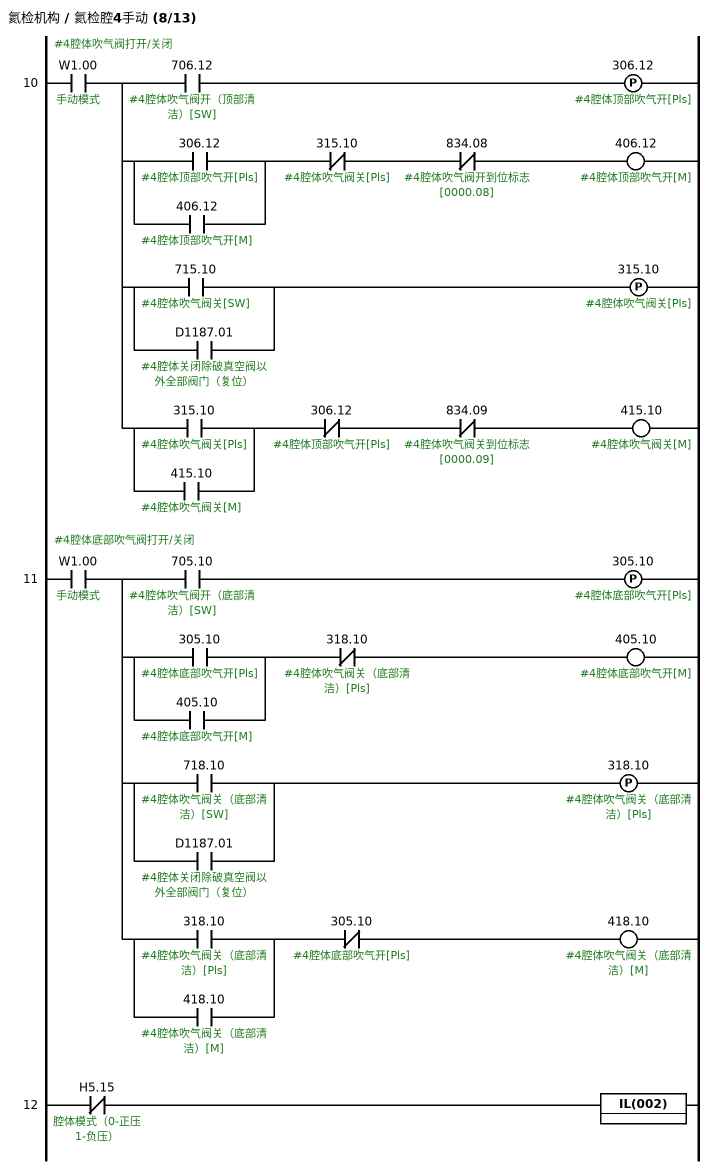
; [picture p216: 氦检机构 / 氦检腔4手动, rungs 10-12]
; rung 10: #4腔体吹气阀打开/关闭
LD W1.00  ; 手动模式
OUT TR0
AND 706.12  ; #4腔体吹气阀开（顶部清洁）[SW]
DIFU(013) 306.12  ; #4腔体顶部吹气开[Pls]
LD TR0
LD 306.12  ; #4腔体顶部吹气开[Pls]
OR 406.12  ; #4腔体顶部吹气开[M]
ANDLD
ANDNOT 315.10  ; #4腔体吹气阀关[Pls]
ANDNOT 834.08  ; #4腔体吹气阀开到位标志[0000.08]
OUT 406.12  ; #4腔体顶部吹气开[M]
LD TR0
LD 715.10  ; #4腔体吹气阀关[SW]
OR D1187.01  ; #4腔体关闭除破真空阀以外全部阀门（复位）
ANDLD
DIFU(013) 315.10  ; #4腔体吹气阀关[Pls]
LD TR0
LD 315.10  ; #4腔体吹气阀关[Pls]
OR 415.10  ; #4腔体吹气阀关[M]
ANDLD
ANDNOT 306.12  ; #4腔体顶部吹气开[Pls]
ANDNOT 834.09  ; #4腔体吹气阀关到位标志[0000.09]
OUT 415.10  ; #4腔体吹气阀关[M]
; rung 11: #4腔体底部吹气阀打开/关闭
LD W1.00  ; 手动模式
OUT TR0
AND 705.10  ; #4腔体吹气阀开（底部清洁）[SW]
DIFU(013) 305.10  ; #4腔体底部吹气开[Pls]
LD TR0
LD 305.10  ; #4腔体底部吹气开[Pls]
OR 405.10  ; #4腔体底部吹气开[M]
ANDLD
ANDNOT 318.10  ; #4腔体吹气阀关（底部清洁）[Pls]
OUT 405.10  ; #4腔体底部吹气开[M]
LD TR0
LD 718.10  ; #4腔体吹气阀关（底部清洁）[SW]
OR D1187.01  ; #4腔体关闭除破真空阀以外全部阀门（复位）
ANDLD
DIFU(013) 318.10  ; #4腔体吹气阀关（底部清洁）[Pls]
LD TR0
LD 318.10  ; #4腔体吹气阀关（底部清洁）[Pls]
OR 418.10  ; #4腔体吹气阀关（底部清洁）[M]
ANDLD
ANDNOT 305.10  ; #4腔体底部吹气开[Pls]
OUT 418.10  ; #4腔体吹气阀关（底部清洁）[M]
; rung 12
LDNOT H5.15  ; 腔体模式（0-正压 1-负压）
IL(002)

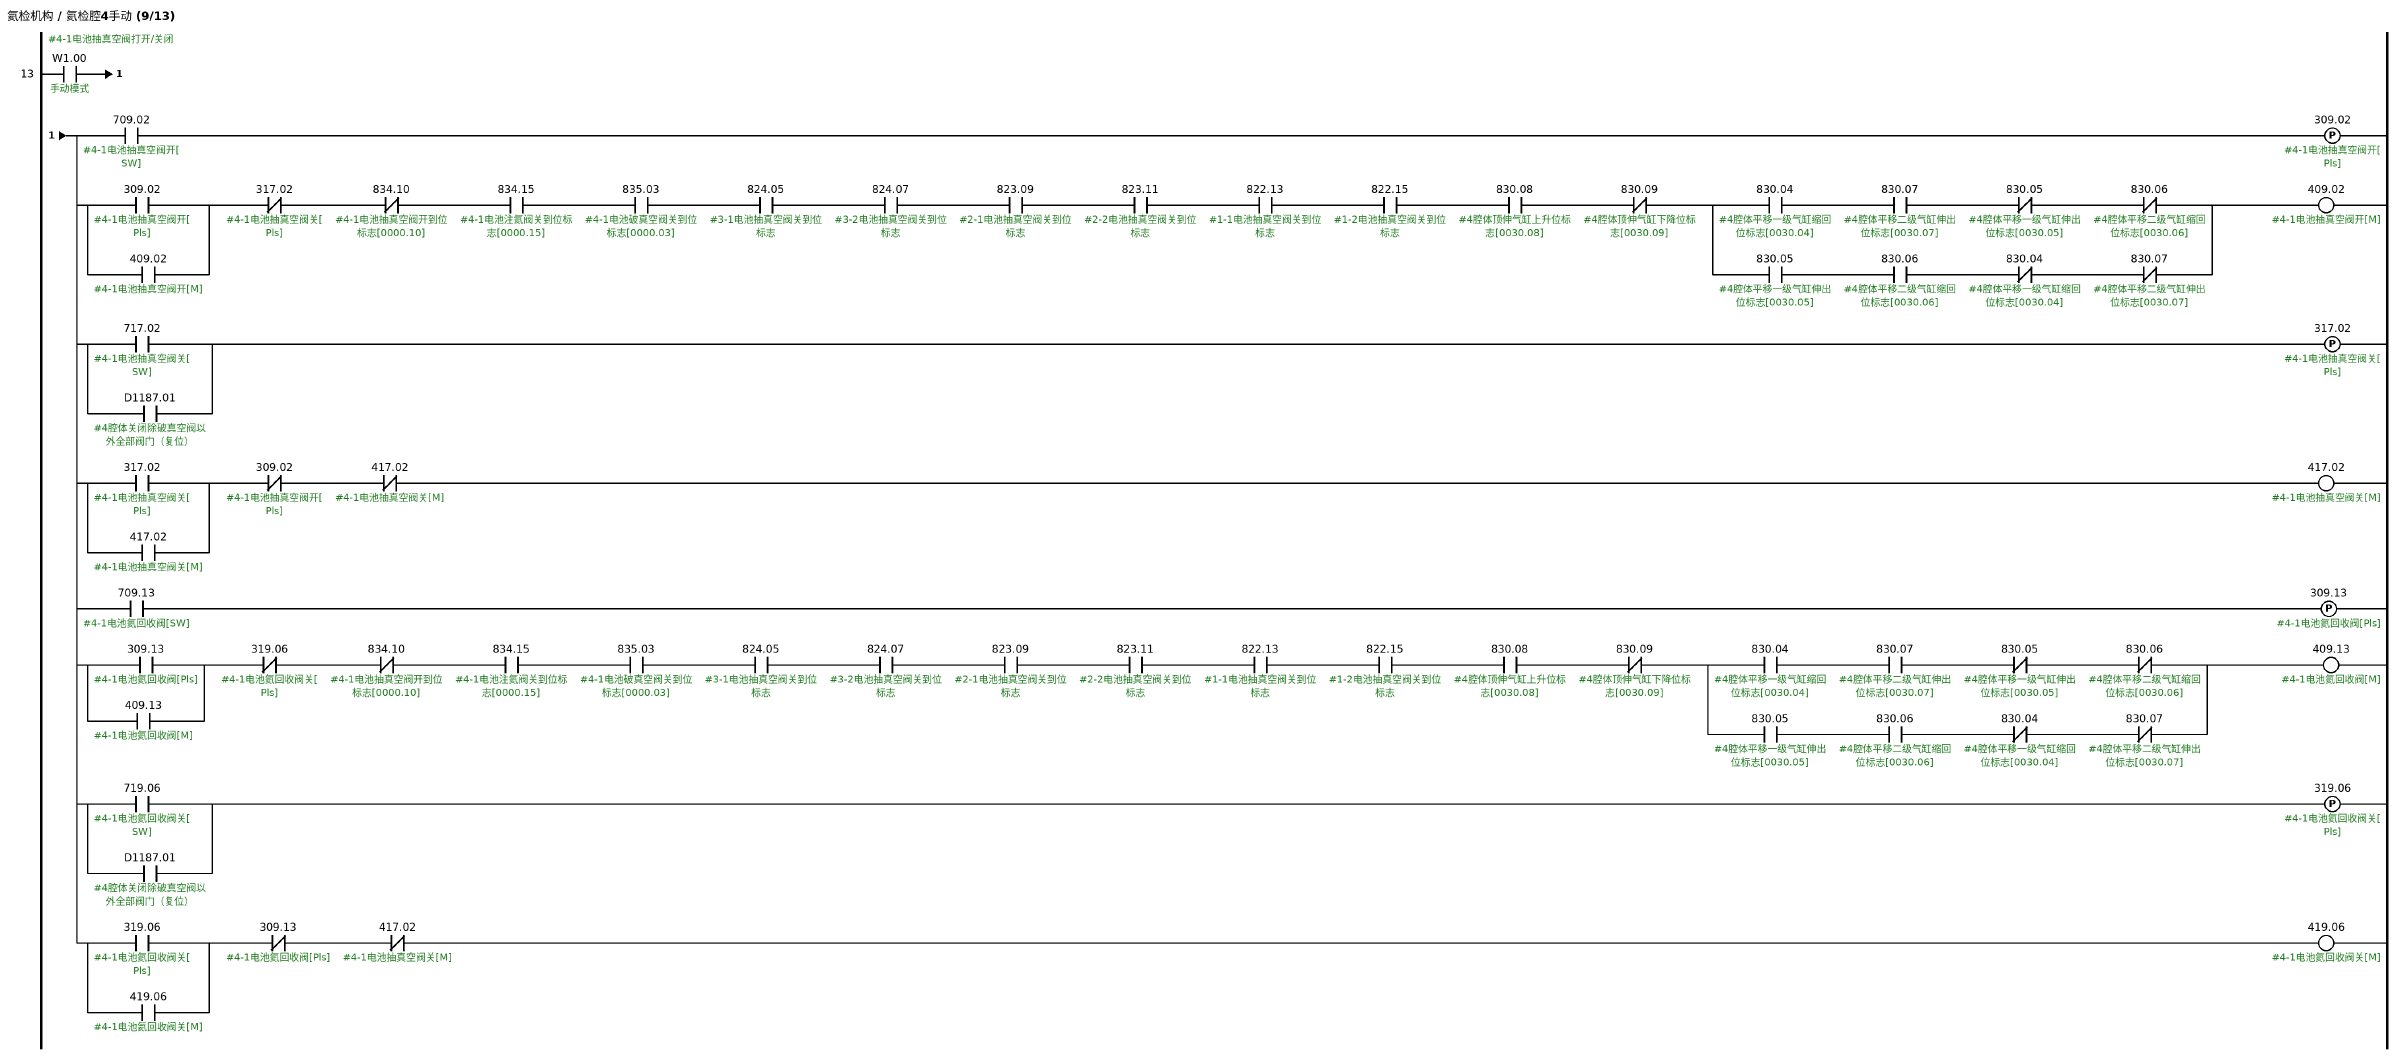
; rung 13: #4-1电池抽真空阀打开/关闭
LD W1.00  ; 手动模式
OUT TR0
AND 709.02  ; #4-1电池抽真空阀开[SW]
DIFU(013) 309.02  ; #4-1电池抽真空阀开[Pls]
LD TR0
LD 309.02  ; #4-1电池抽真空阀开[Pls]
OR 409.02  ; #4-1电池抽真空阀开[M]
ANDLD
ANDNOT 317.02  ; #4-1电池抽真空阀关[Pls]
ANDNOT 834.10  ; #4-1电池抽真空阀开到位标志[0000.10]
AND 834.15  ; #4-1电池注氦阀关到位标志[0000.15]
AND 835.03  ; #4-1电池破真空阀关到位标志[0000.03]
AND 824.05  ; #3-1电池抽真空阀关到位标志
AND 824.07  ; #3-2电池抽真空阀关到位标志
AND 823.09  ; #2-1电池抽真空阀关到位标志
AND 823.11  ; #2-2电池抽真空阀关到位标志
AND 822.13  ; #1-1电池抽真空阀关到位标志
AND 822.15  ; #1-2电池抽真空阀关到位标志
AND 830.08  ; #4腔体顶伸气缸上升位标志[0030.08]
ANDNOT 830.09  ; #4腔体顶伸气缸下降位标志[0030.09]
LD 830.04  ; #4腔体平移一级气缸缩回位标志[0030.04]
AND 830.07  ; #4腔体平移二级气缸伸出位标志[0030.07]
ANDNOT 830.05  ; #4腔体平移一级气缸伸出位标志[0030.05]
ANDNOT 830.06  ; #4腔体平移二级气缸缩回位标志[0030.06]
LD 830.05  ; #4腔体平移一级气缸伸出位标志[0030.05]
AND 830.06  ; #4腔体平移二级气缸缩回位标志[0030.06]
ANDNOT 830.04  ; #4腔体平移一级气缸缩回位标志[0030.04]
ANDNOT 830.07  ; #4腔体平移二级气缸伸出位标志[0030.07]
ORLD
ANDLD
OUT 409.02  ; #4-1电池抽真空阀开[M]
LD TR0
LD 717.02  ; #4-1电池抽真空阀关[SW]
OR D1187.01  ; #4腔体关闭除破真空阀以外全部阀门（复位）
ANDLD
DIFU(013) 317.02  ; #4-1电池抽真空阀关[Pls]
LD TR0
LD 317.02  ; #4-1电池抽真空阀关[Pls]
OR 417.02  ; #4-1电池抽真空阀关[M]
ANDLD
ANDNOT 309.02  ; #4-1电池抽真空阀开[Pls]
ANDNOT 417.02  ; #4-1电池抽真空阀关[M]
OUT 417.02  ; #4-1电池抽真空阀关[M]
LD TR0
AND 709.13  ; #4-1电池氦回收阀[SW]
DIFU(013) 309.13  ; #4-1电池氦回收阀[Pls]
LD TR0
LD 309.13  ; #4-1电池氦回收阀[Pls]
OR 409.13  ; #4-1电池氦回收阀[M]
ANDLD
ANDNOT 319.06  ; #4-1电池氦回收阀关[Pls]
ANDNOT 834.10  ; #4-1电池抽真空阀开到位标志[0000.10]
AND 834.15  ; #4-1电池注氦阀关到位标志[0000.15]
AND 835.03  ; #4-1电池破真空阀关到位标志[0000.03]
AND 824.05  ; #3-1电池抽真空阀关到位标志
AND 824.07  ; #3-2电池抽真空阀关到位标志
AND 823.09  ; #2-1电池抽真空阀关到位标志
AND 823.11  ; #2-2电池抽真空阀关到位标志
AND 822.13  ; #1-1电池抽真空阀关到位标志
AND 822.15  ; #1-2电池抽真空阀关到位标志
AND 830.08  ; #4腔体顶伸气缸上升位标志[0030.08]
ANDNOT 830.09  ; #4腔体顶伸气缸下降位标志[0030.09]
LD 830.04  ; #4腔体平移一级气缸缩回位标志[0030.04]
AND 830.07  ; #4腔体平移二级气缸伸出位标志[0030.07]
ANDNOT 830.05  ; #4腔体平移一级气缸伸出位标志[0030.05]
ANDNOT 830.06  ; #4腔体平移二级气缸缩回位标志[0030.06]
LD 830.05  ; #4腔体平移一级气缸伸出位标志[0030.05]
AND 830.06  ; #4腔体平移二级气缸缩回位标志[0030.06]
ANDNOT 830.04  ; #4腔体平移一级气缸缩回位标志[0030.04]
ANDNOT 830.07  ; #4腔体平移二级气缸伸出位标志[0030.07]
ORLD
ANDLD
OUT 409.13  ; #4-1电池氦回收阀[M]
LD TR0
LD 719.06  ; #4-1电池氦回收阀关[SW]
OR D1187.01  ; #4腔体关闭除破真空阀以外全部阀门（复位）
ANDLD
DIFU(013) 319.06  ; #4-1电池氦回收阀关[Pls]
LD TR0
LD 319.06  ; #4-1电池氦回收阀关[Pls]
OR 419.06  ; #4-1电池氦回收阀关[M]
ANDLD
ANDNOT 309.13  ; #4-1电池氦回收阀[Pls]
ANDNOT 417.02  ; #4-1电池抽真空阀关[M]
OUT 419.06  ; #4-1电池氦回收阀关[M]

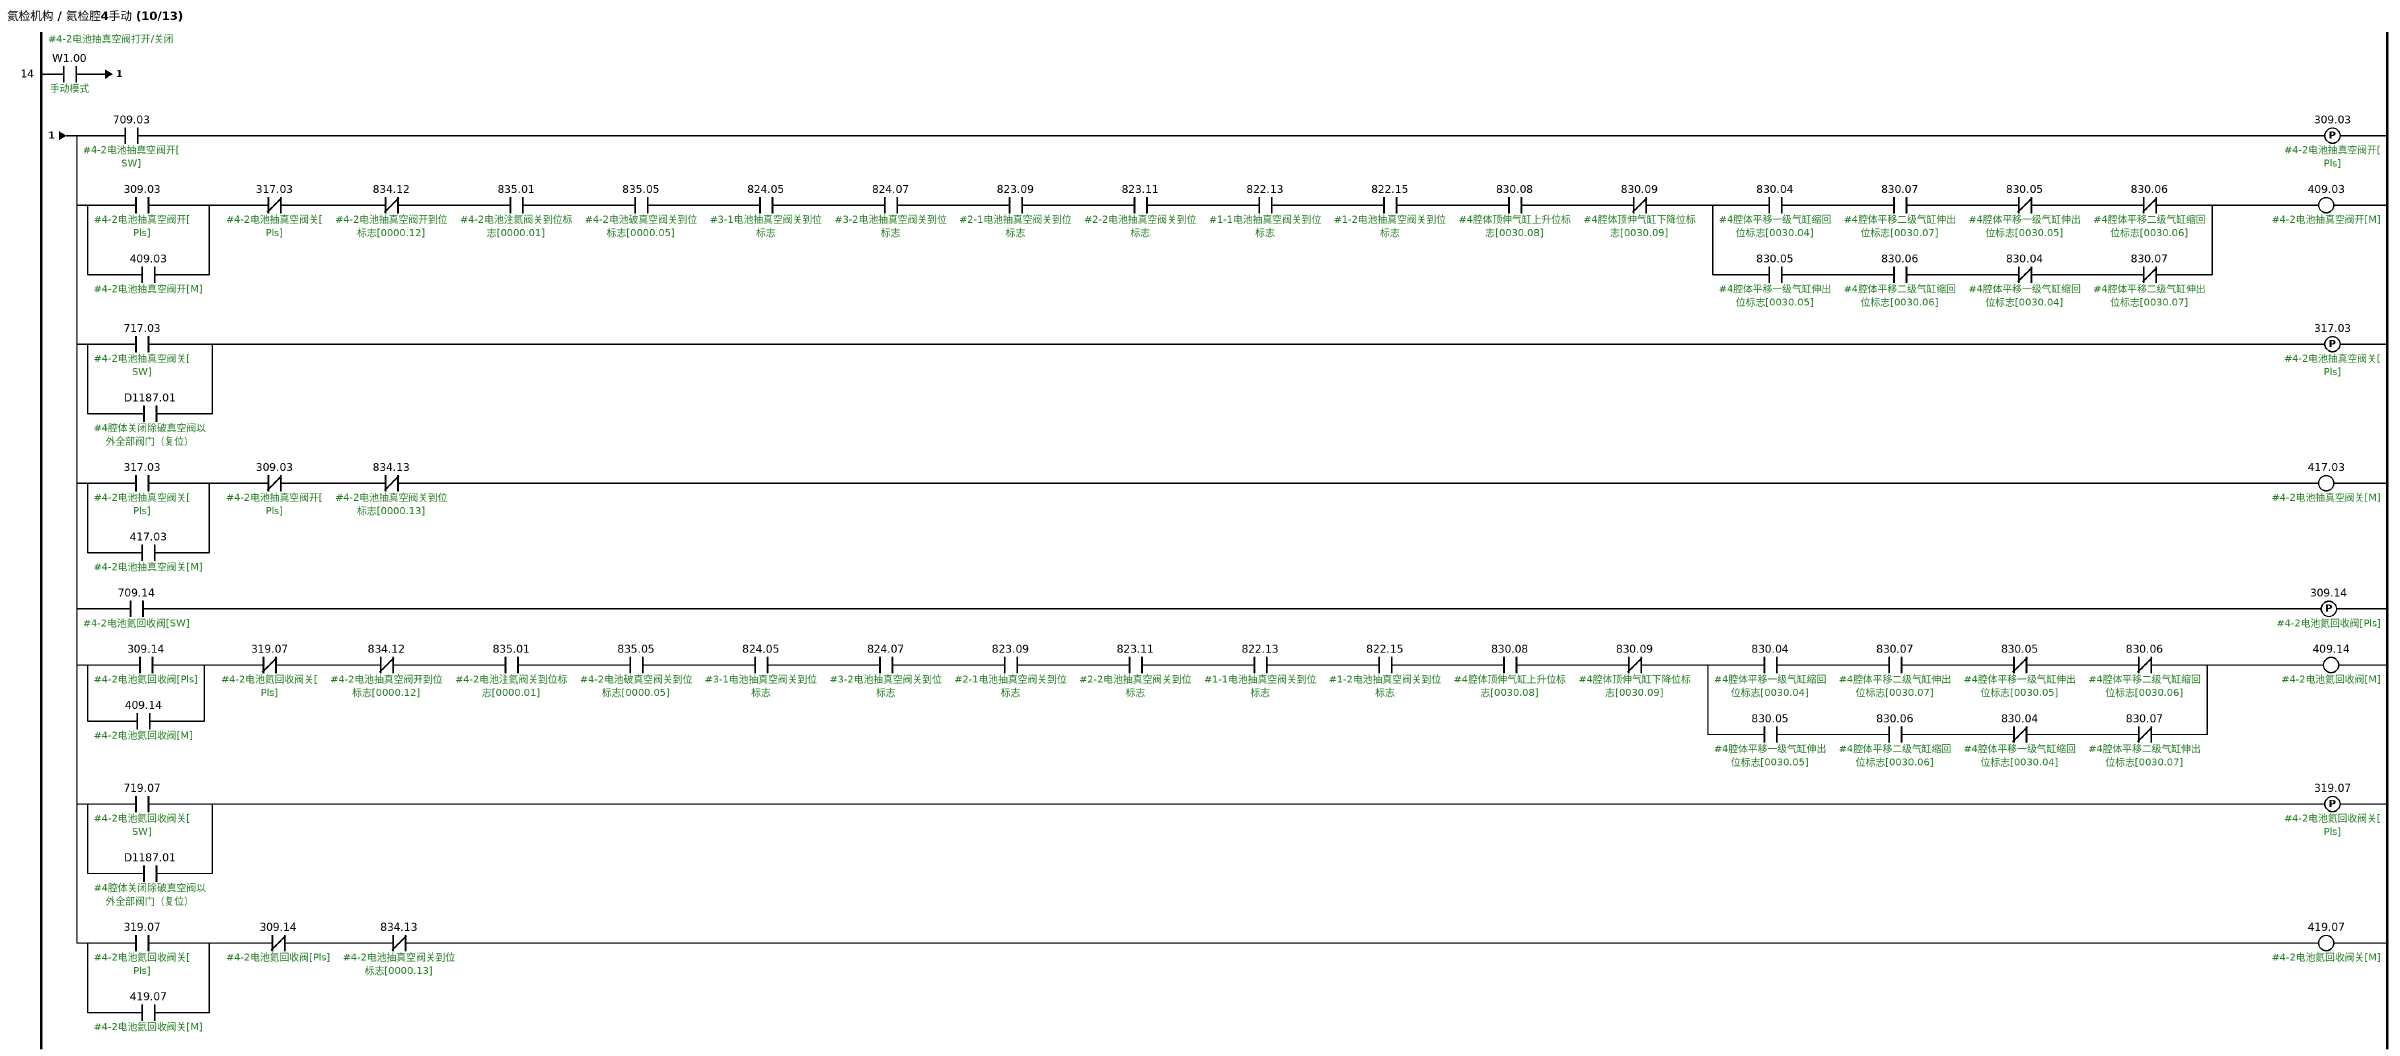
; rung 14: #4-2电池抽真空阀打开/关闭
LD W1.00  ; 手动模式
OUT TR0
AND 709.03  ; #4-2电池抽真空阀开[SW]
DIFU(013) 309.03  ; #4-2电池抽真空阀开[Pls]
LD TR0
LD 309.03  ; #4-2电池抽真空阀开[Pls]
OR 409.03  ; #4-2电池抽真空阀开[M]
ANDLD
ANDNOT 317.03  ; #4-2电池抽真空阀关[Pls]
ANDNOT 834.12  ; #4-2电池抽真空阀开到位标志[0000.12]
AND 835.01  ; #4-2电池注氦阀关到位标志[0000.01]
AND 835.05  ; #4-2电池破真空阀关到位标志[0000.05]
AND 824.05  ; #3-1电池抽真空阀关到位标志
AND 824.07  ; #3-2电池抽真空阀关到位标志
AND 823.09  ; #2-1电池抽真空阀关到位标志
AND 823.11  ; #2-2电池抽真空阀关到位标志
AND 822.13  ; #1-1电池抽真空阀关到位标志
AND 822.15  ; #1-2电池抽真空阀关到位标志
AND 830.08  ; #4腔体顶伸气缸上升位标志[0030.08]
ANDNOT 830.09  ; #4腔体顶伸气缸下降位标志[0030.09]
LD 830.04  ; #4腔体平移一级气缸缩回位标志[0030.04]
AND 830.07  ; #4腔体平移二级气缸伸出位标志[0030.07]
ANDNOT 830.05  ; #4腔体平移一级气缸伸出位标志[0030.05]
ANDNOT 830.06  ; #4腔体平移二级气缸缩回位标志[0030.06]
LD 830.05  ; #4腔体平移一级气缸伸出位标志[0030.05]
AND 830.06  ; #4腔体平移二级气缸缩回位标志[0030.06]
ANDNOT 830.04  ; #4腔体平移一级气缸缩回位标志[0030.04]
ANDNOT 830.07  ; #4腔体平移二级气缸伸出位标志[0030.07]
ORLD
ANDLD
OUT 409.03  ; #4-2电池抽真空阀开[M]
LD TR0
LD 717.03  ; #4-2电池抽真空阀关[SW]
OR D1187.01  ; #4腔体关闭除破真空阀以外全部阀门（复位）
ANDLD
DIFU(013) 317.03  ; #4-2电池抽真空阀关[Pls]
LD TR0
LD 317.03  ; #4-2电池抽真空阀关[Pls]
OR 417.03  ; #4-2电池抽真空阀关[M]
ANDLD
ANDNOT 309.03  ; #4-2电池抽真空阀开[Pls]
ANDNOT 834.13  ; #4-2电池抽真空阀关到位标志[0000.13]
OUT 417.03  ; #4-2电池抽真空阀关[M]
LD TR0
AND 709.14  ; #4-2电池氦回收阀[SW]
DIFU(013) 309.14  ; #4-2电池氦回收阀[Pls]
LD TR0
LD 309.14  ; #4-2电池氦回收阀[Pls]
OR 409.14  ; #4-2电池氦回收阀[M]
ANDLD
ANDNOT 319.07  ; #4-2电池氦回收阀关[Pls]
ANDNOT 834.12  ; #4-2电池抽真空阀开到位标志[0000.12]
AND 835.01  ; #4-2电池注氦阀关到位标志[0000.01]
AND 835.05  ; #4-2电池破真空阀关到位标志[0000.05]
AND 824.05  ; #3-1电池抽真空阀关到位标志
AND 824.07  ; #3-2电池抽真空阀关到位标志
AND 823.09  ; #2-1电池抽真空阀关到位标志
AND 823.11  ; #2-2电池抽真空阀关到位标志
AND 822.13  ; #1-1电池抽真空阀关到位标志
AND 822.15  ; #1-2电池抽真空阀关到位标志
AND 830.08  ; #4腔体顶伸气缸上升位标志[0030.08]
ANDNOT 830.09  ; #4腔体顶伸气缸下降位标志[0030.09]
LD 830.04  ; #4腔体平移一级气缸缩回位标志[0030.04]
AND 830.07  ; #4腔体平移二级气缸伸出位标志[0030.07]
ANDNOT 830.05  ; #4腔体平移一级气缸伸出位标志[0030.05]
ANDNOT 830.06  ; #4腔体平移二级气缸缩回位标志[0030.06]
LD 830.05  ; #4腔体平移一级气缸伸出位标志[0030.05]
AND 830.06  ; #4腔体平移二级气缸缩回位标志[0030.06]
ANDNOT 830.04  ; #4腔体平移一级气缸缩回位标志[0030.04]
ANDNOT 830.07  ; #4腔体平移二级气缸伸出位标志[0030.07]
ORLD
ANDLD
OUT 409.14  ; #4-2电池氦回收阀[M]
LD TR0
LD 719.07  ; #4-2电池氦回收阀关[SW]
OR D1187.01  ; #4腔体关闭除破真空阀以外全部阀门（复位）
ANDLD
DIFU(013) 319.07  ; #4-2电池氦回收阀关[Pls]
LD TR0
LD 319.07  ; #4-2电池氦回收阀关[Pls]
OR 419.07  ; #4-2电池氦回收阀关[M]
ANDLD
ANDNOT 309.14  ; #4-2电池氦回收阀[Pls]
ANDNOT 834.13  ; #4-2电池抽真空阀关到位标志[0000.13]
OUT 419.07  ; #4-2电池氦回收阀关[M]

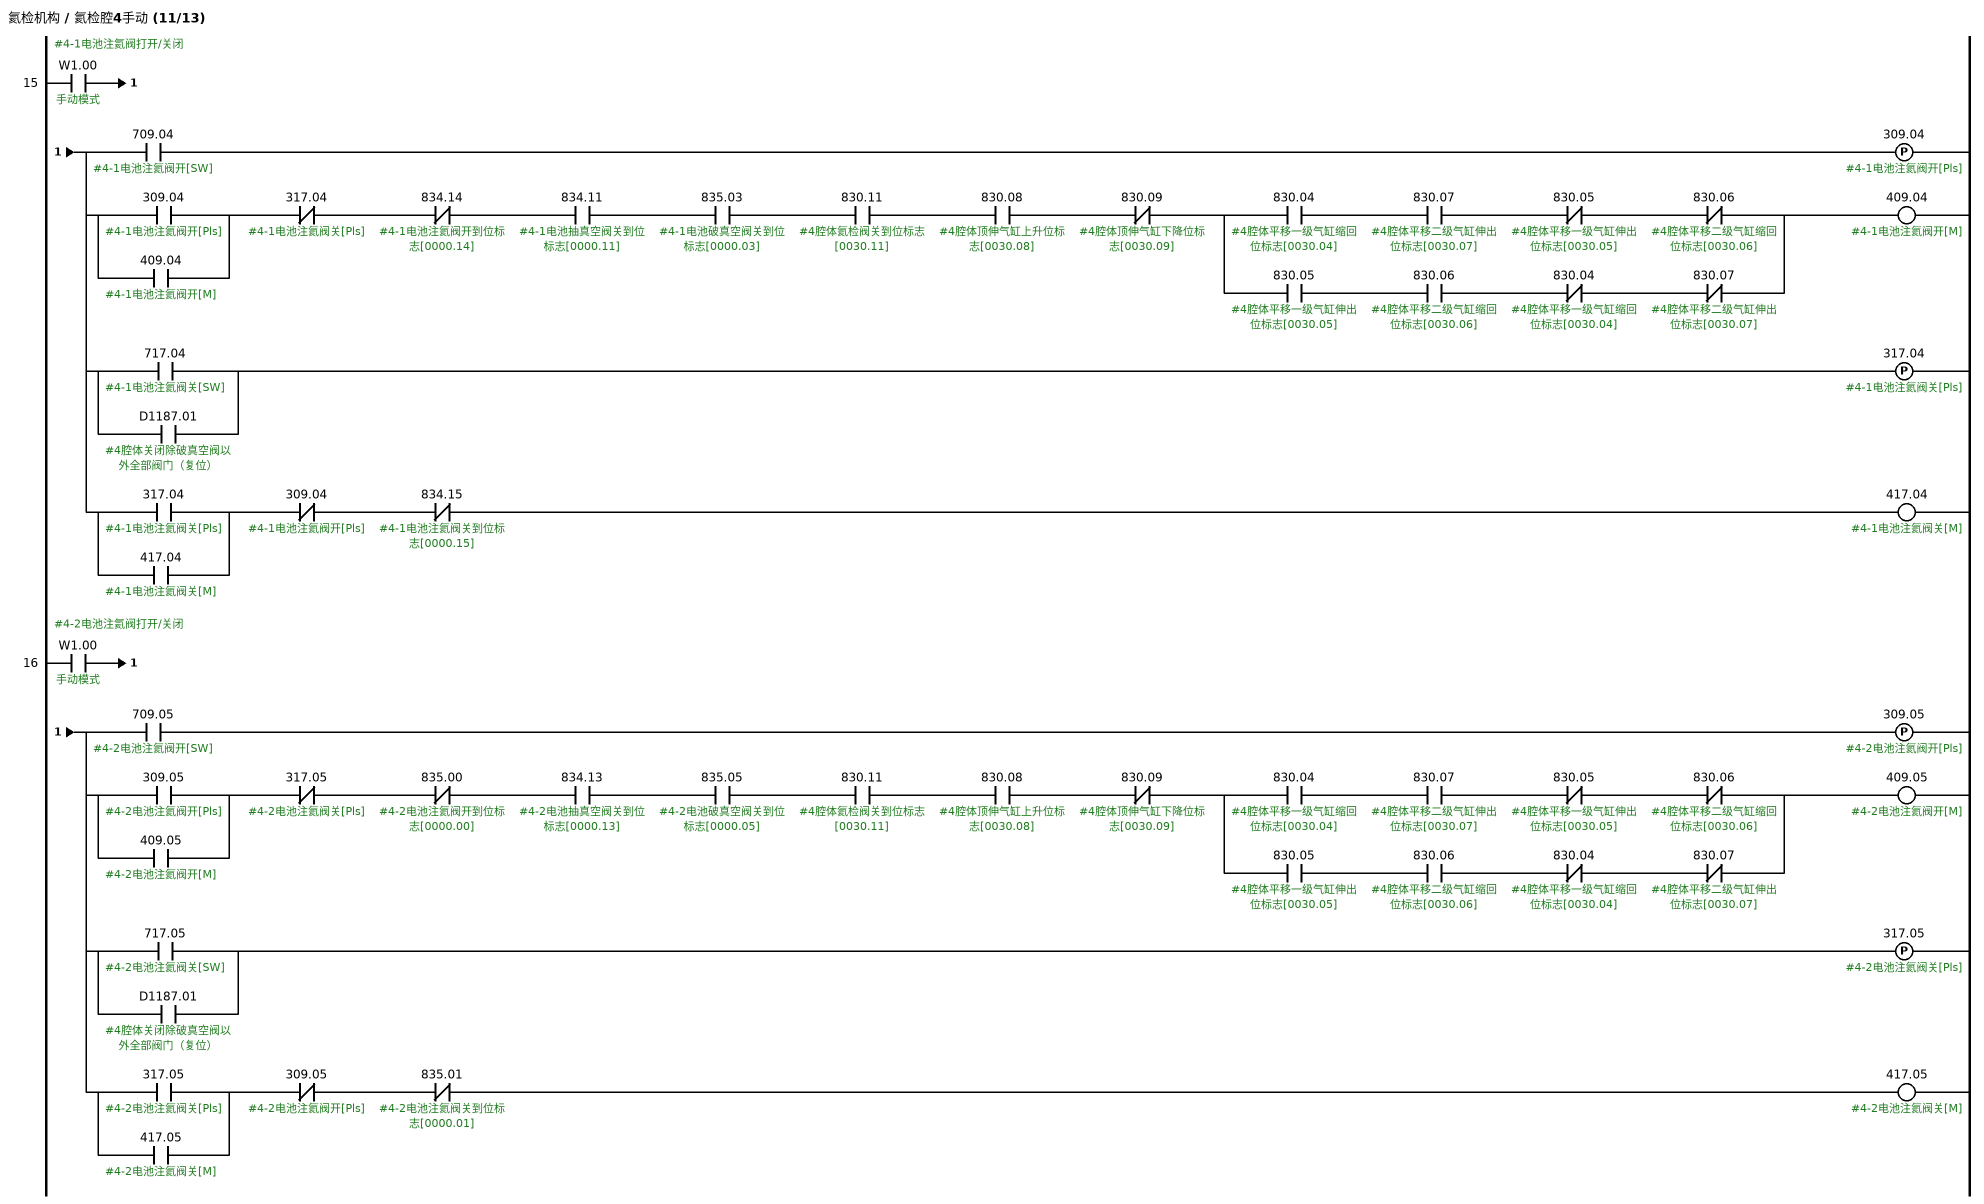
; rung 15: #4-1电池注氦阀打开/关闭
LD W1.00  ; 手动模式
OUT TR0
AND 709.04  ; #4-1电池注氦阀开[SW]
DIFU(013) 309.04  ; #4-1电池注氦阀开[Pls]
LD TR0
LD 309.04  ; #4-1电池注氦阀开[Pls]
OR 409.04  ; #4-1电池注氦阀开[M]
ANDLD
ANDNOT 317.04  ; #4-1电池注氦阀关[Pls]
ANDNOT 834.14  ; #4-1电池注氦阀开到位标志[0000.14]
AND 834.11  ; #4-1电池抽真空阀关到位标志[0000.11]
AND 835.03  ; #4-1电池破真空阀关到位标志[0000.03]
AND 830.11  ; #4腔体氦检阀关到位标志[0030.11]
AND 830.08  ; #4腔体顶伸气缸上升位标志[0030.08]
ANDNOT 830.09  ; #4腔体顶伸气缸下降位标志[0030.09]
LD 830.04  ; #4腔体平移一级气缸缩回位标志[0030.04]
AND 830.07  ; #4腔体平移二级气缸伸出位标志[0030.07]
ANDNOT 830.05  ; #4腔体平移一级气缸伸出位标志[0030.05]
ANDNOT 830.06  ; #4腔体平移二级气缸缩回位标志[0030.06]
LD 830.05  ; #4腔体平移一级气缸伸出位标志[0030.05]
AND 830.06  ; #4腔体平移二级气缸缩回位标志[0030.06]
ANDNOT 830.04  ; #4腔体平移一级气缸缩回位标志[0030.04]
ANDNOT 830.07  ; #4腔体平移二级气缸伸出位标志[0030.07]
ORLD
ANDLD
OUT 409.04  ; #4-1电池注氦阀开[M]
LD TR0
LD 717.04  ; #4-1电池注氦阀关[SW]
OR D1187.01  ; #4腔体关闭除破真空阀以外全部阀门（复位）
ANDLD
DIFU(013) 317.04  ; #4-1电池注氦阀关[Pls]
LD TR0
LD 317.04  ; #4-1电池注氦阀关[Pls]
OR 417.04  ; #4-1电池注氦阀关[M]
ANDLD
ANDNOT 309.04  ; #4-1电池注氦阀开[Pls]
ANDNOT 834.15  ; #4-1电池注氦阀关到位标志[0000.15]
OUT 417.04  ; #4-1电池注氦阀关[M]
; rung 16: #4-2电池注氦阀打开/关闭
LD W1.00  ; 手动模式
OUT TR0
AND 709.05  ; #4-2电池注氦阀开[SW]
DIFU(013) 309.05  ; #4-2电池注氦阀开[Pls]
LD TR0
LD 309.05  ; #4-2电池注氦阀开[Pls]
OR 409.05  ; #4-2电池注氦阀开[M]
ANDLD
ANDNOT 317.05  ; #4-2电池注氦阀关[Pls]
ANDNOT 835.00  ; #4-2电池注氦阀开到位标志[0000.00]
AND 834.13  ; #4-2电池抽真空阀关到位标志[0000.13]
AND 835.05  ; #4-2电池破真空阀关到位标志[0000.05]
AND 830.11  ; #4腔体氦检阀关到位标志[0030.11]
AND 830.08  ; #4腔体顶伸气缸上升位标志[0030.08]
ANDNOT 830.09  ; #4腔体顶伸气缸下降位标志[0030.09]
LD 830.04  ; #4腔体平移一级气缸缩回位标志[0030.04]
AND 830.07  ; #4腔体平移二级气缸伸出位标志[0030.07]
ANDNOT 830.05  ; #4腔体平移一级气缸伸出位标志[0030.05]
ANDNOT 830.06  ; #4腔体平移二级气缸缩回位标志[0030.06]
LD 830.05  ; #4腔体平移一级气缸伸出位标志[0030.05]
AND 830.06  ; #4腔体平移二级气缸缩回位标志[0030.06]
ANDNOT 830.04  ; #4腔体平移一级气缸缩回位标志[0030.04]
ANDNOT 830.07  ; #4腔体平移二级气缸伸出位标志[0030.07]
ORLD
ANDLD
OUT 409.05  ; #4-2电池注氦阀开[M]
LD TR0
LD 717.05  ; #4-2电池注氦阀关[SW]
OR D1187.01  ; #4腔体关闭除破真空阀以外全部阀门（复位）
ANDLD
DIFU(013) 317.05  ; #4-2电池注氦阀关[Pls]
LD TR0
LD 317.05  ; #4-2电池注氦阀关[Pls]
OR 417.05  ; #4-2电池注氦阀关[M]
ANDLD
ANDNOT 309.05  ; #4-2电池注氦阀开[Pls]
ANDNOT 835.01  ; #4-2电池注氦阀关到位标志[0000.01]
OUT 417.05  ; #4-2电池注氦阀关[M]

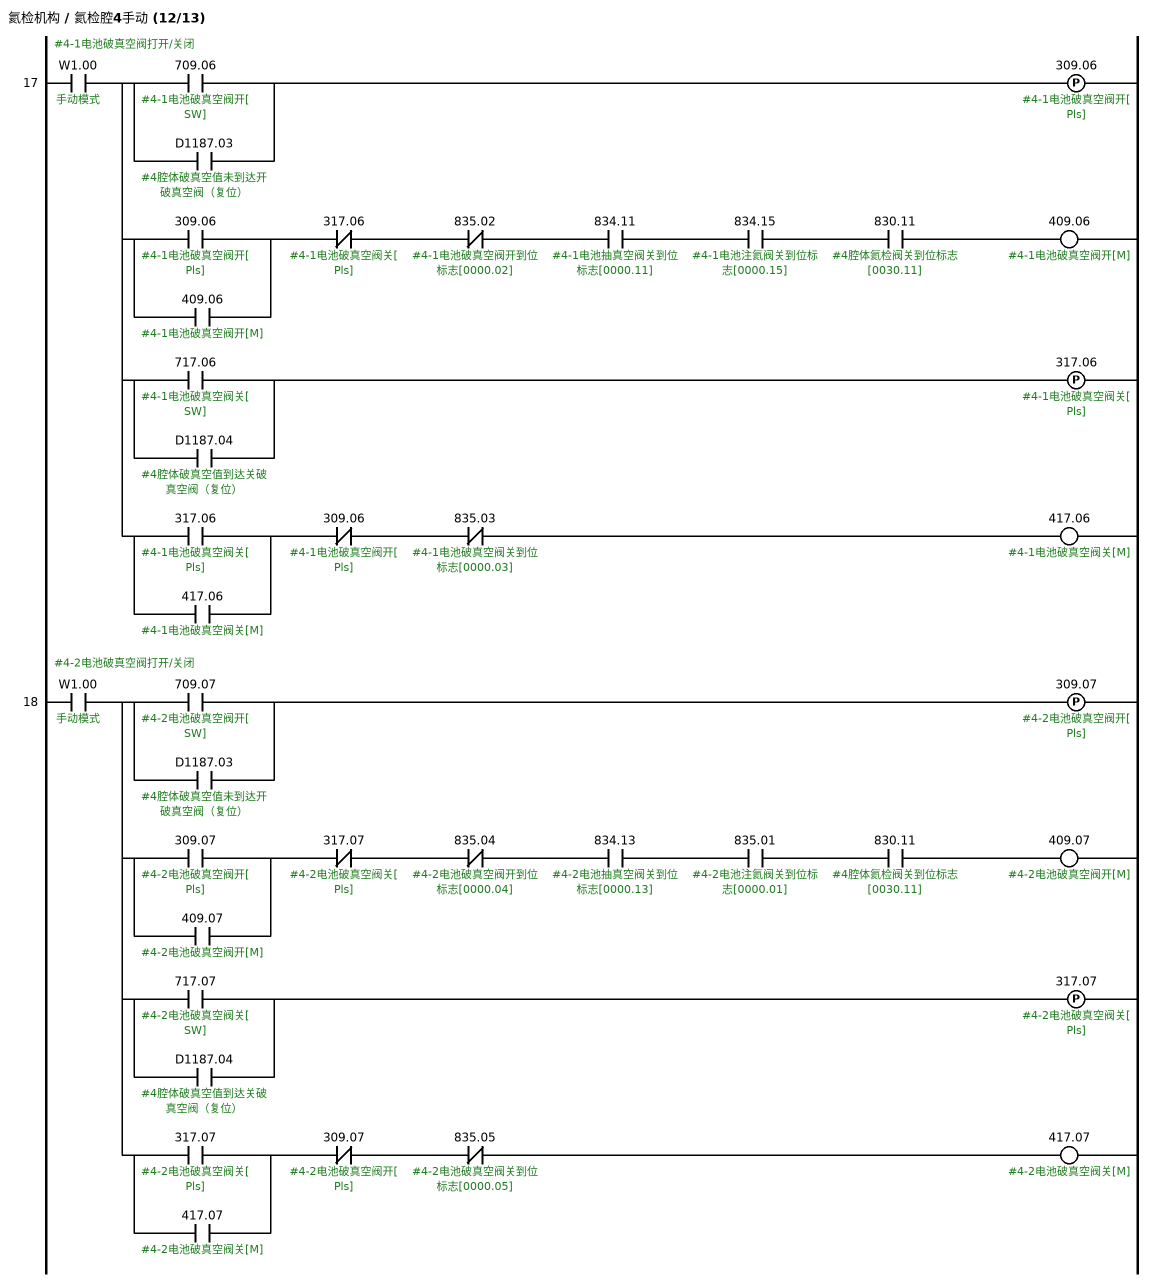
; rung 17: #4-1电池破真空阀打开/关闭
LD W1.00  ; 手动模式
OUT TR0
LD 709.06  ; #4-1电池破真空阀开[SW]
OR D1187.03  ; #4腔体破真空值未到达开破真空阀（复位）
ANDLD
DIFU(013) 309.06  ; #4-1电池破真空阀开[Pls]
LD TR0
LD 309.06  ; #4-1电池破真空阀开[Pls]
OR 409.06  ; #4-1电池破真空阀开[M]
ANDLD
ANDNOT 317.06  ; #4-1电池破真空阀关[Pls]
ANDNOT 835.02  ; #4-1电池破真空阀开到位标志[0000.02]
AND 834.11  ; #4-1电池抽真空阀关到位标志[0000.11]
AND 834.15  ; #4-1电池注氦阀关到位标志[0000.15]
AND 830.11  ; #4腔体氦检阀关到位标志[0030.11]
OUT 409.06  ; #4-1电池破真空阀开[M]
LD TR0
LD 717.06  ; #4-1电池破真空阀关[SW]
OR D1187.04  ; #4腔体破真空值到达关破真空阀（复位）
ANDLD
DIFU(013) 317.06  ; #4-1电池破真空阀关[Pls]
LD TR0
LD 317.06  ; #4-1电池破真空阀关[Pls]
OR 417.06  ; #4-1电池破真空阀关[M]
ANDLD
ANDNOT 309.06  ; #4-1电池破真空阀开[Pls]
ANDNOT 835.03  ; #4-1电池破真空阀关到位标志[0000.03]
OUT 417.06  ; #4-1电池破真空阀关[M]
; rung 18: #4-2电池破真空阀打开/关闭
LD W1.00  ; 手动模式
OUT TR0
LD 709.07  ; #4-2电池破真空阀开[SW]
OR D1187.03  ; #4腔体破真空值未到达开破真空阀（复位）
ANDLD
DIFU(013) 309.07  ; #4-2电池破真空阀开[Pls]
LD TR0
LD 309.07  ; #4-2电池破真空阀开[Pls]
OR 409.07  ; #4-2电池破真空阀开[M]
ANDLD
ANDNOT 317.07  ; #4-2电池破真空阀关[Pls]
ANDNOT 835.04  ; #4-2电池破真空阀开到位标志[0000.04]
AND 834.13  ; #4-2电池抽真空阀关到位标志[0000.13]
AND 835.01  ; #4-2电池注氦阀关到位标志[0000.01]
AND 830.11  ; #4腔体氦检阀关到位标志[0030.11]
OUT 409.07  ; #4-2电池破真空阀开[M]
LD TR0
LD 717.07  ; #4-2电池破真空阀关[SW]
OR D1187.04  ; #4腔体破真空值到达关破真空阀（复位）
ANDLD
DIFU(013) 317.07  ; #4-2电池破真空阀关[Pls]
LD TR0
LD 317.07  ; #4-2电池破真空阀关[Pls]
OR 417.07  ; #4-2电池破真空阀关[M]
ANDLD
ANDNOT 309.07  ; #4-2电池破真空阀开[Pls]
ANDNOT 835.05  ; #4-2电池破真空阀关到位标志[0000.05]
OUT 417.07  ; #4-2电池破真空阀关[M]

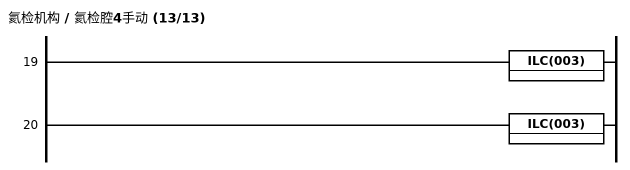
; rung 19
ILC(003)
; rung 20
ILC(003)

### Section 氦检腔1自动

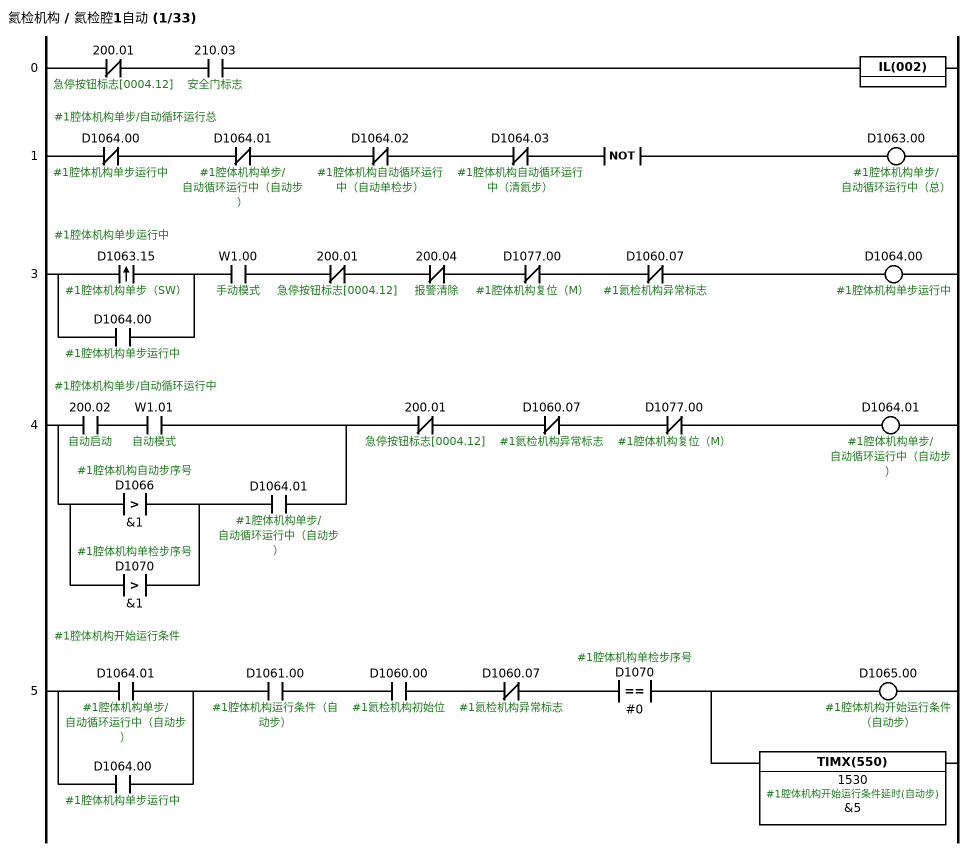
; rung 0
LDNOT 200.01  ; 急停按钮标志[0004.12]
AND 210.03  ; 安全门标志
IL(002)
; rung 1: #1腔体机构单步/自动循环运行总
LDNOT D1064.00  ; #1腔体机构单步运行中
ANDNOT D1064.01  ; #1腔体机构单步/自动循环运行中（自动步）
ANDNOT D1064.02  ; #1腔体机构自动循环运行中（自动单检步）
ANDNOT D1064.03  ; #1腔体机构自动循环运行中（清氦步）
NOT(520)
OUT D1063.00  ; #1腔体机构单步/自动循环运行中（总）
; rung 2: ******************************* / 自动双检步序 / *******************************
; rung 3: #1腔体机构单步运行中
@LD D1063.15  ; #1腔体机构单步（SW）
OR D1064.00  ; #1腔体机构单步运行中
AND W1.00  ; 手动模式
ANDNOT 200.01  ; 急停按钮标志[0004.12]
ANDNOT 200.04  ; 报警清除
ANDNOT D1077.00  ; #1腔体机构复位（M）
ANDNOT D1060.07  ; #1氦检机构异常标志
OUT D1064.00  ; #1腔体机构单步运行中
; rung 4: #1腔体机构单步/自动循环运行中
LD 200.02  ; 自动启动
AND W1.01  ; 自动模式
LD>L(321) D1066 &1  ; #1腔体机构自动步序号
OR>L(321) D1070 &1  ; #1腔体机构单检步序号
AND D1064.01  ; #1腔体机构单步/自动循环运行中（自动步）
ORLD
ANDNOT 200.01  ; 急停按钮标志[0004.12]
ANDNOT D1060.07  ; #1氦检机构异常标志
ANDNOT D1077.00  ; #1腔体机构复位（M）
OUT D1064.01  ; #1腔体机构单步/自动循环运行中（自动步）
; rung 5: #1腔体机构开始运行条件
LD D1064.01  ; #1腔体机构单步/自动循环运行中（自动步）
OR D1064.00  ; #1腔体机构单步运行中
AND D1061.00  ; #1腔体机构运行条件（自动步）
AND D1060.00  ; #1氦检机构初始位
ANDNOT D1060.07  ; #1氦检机构异常标志
AND=L(301) D1070 #0  ; #1腔体机构单检步序号
OUT D1065.00  ; #1腔体机构开始运行条件（自动步）
TIMX(550) 1530 &5  ; #1腔体机构开始运行条件延时(自动步)

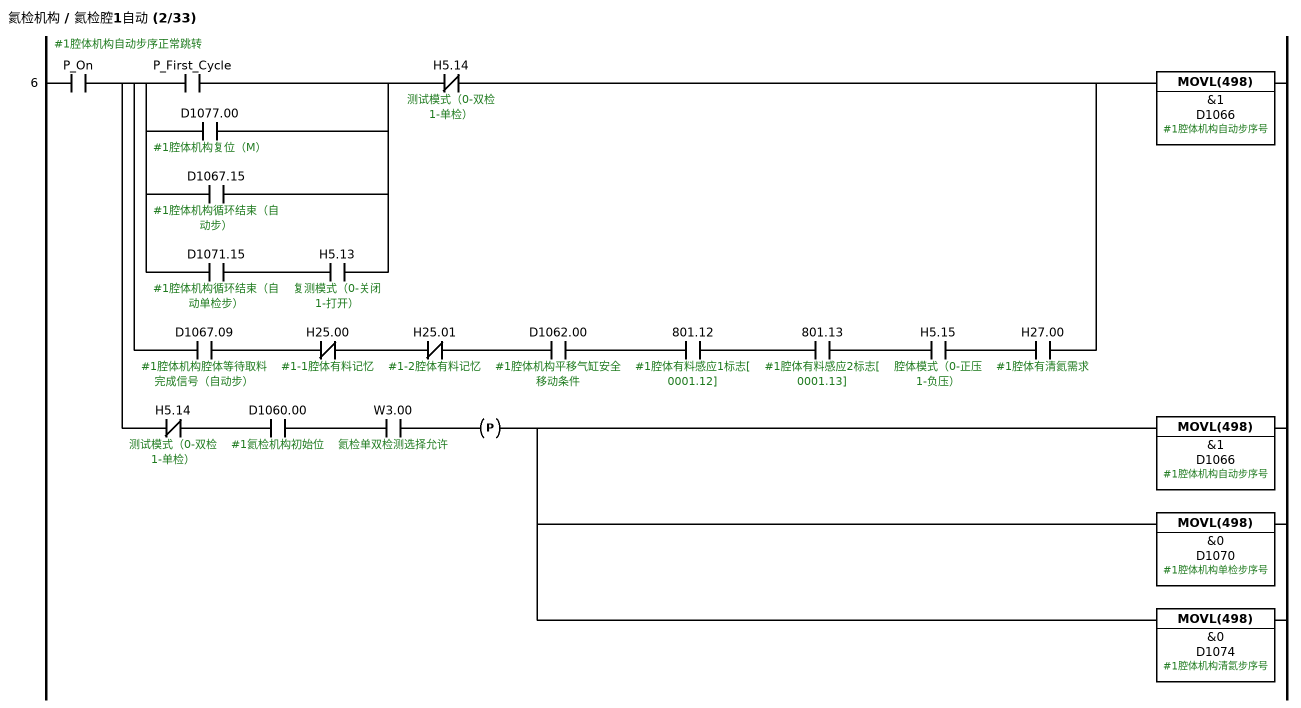
; rung 6: #1腔体机构自动步序正常跳转
LD P_On
OUT TR0
LD P_First_Cycle
OR D1077.00  ; #1腔体机构复位（M）
OR D1067.15  ; #1腔体机构循环结束（自动步）
LD D1071.15  ; #1腔体机构循环结束（自动单检步）
AND H5.13  ; 复测模式（0-关闭 1-打开）
ORLD
ANDNOT H5.14  ; 测试模式（0-双检 1-单检）
LD D1067.09  ; #1腔体机构腔体等待取料完成信号（自动步）  // 负压有清氦需求时，无需回初始位,直接跳回初始步序（D1066.00）
ANDNOT H25.00  ; #1-1腔体有料记忆
ANDNOT H25.01  ; #1-2腔体有料记忆
AND D1062.00  ; #1腔体机构平移气缸安全移动条件
AND 801.12  ; #1腔体有料感应1标志[0001.12]
AND 801.13  ; #1腔体有料感应2标志[0001.13]
AND H5.15  ; 腔体模式（0-正压 1-负压）
AND H27.00  ; #1腔体有清氦需求
ORLD
ANDLD
MOVL(498) &1 D1066  ; #1腔体机构自动步序号
LD TR0
ANDNOT H5.14  ; 测试模式（0-双检 1-单检）
AND D1060.00  ; #1氦检机构初始位
AND W3.00  ; 氦检单双检测选择允许
UP(521)
MOVL(498) &1 D1066  ; #1腔体机构自动步序号
MOVL(498) &0 D1070  ; #1腔体机构单检步序号
MOVL(498) &0 D1074  ; #1腔体机构清氦步序号

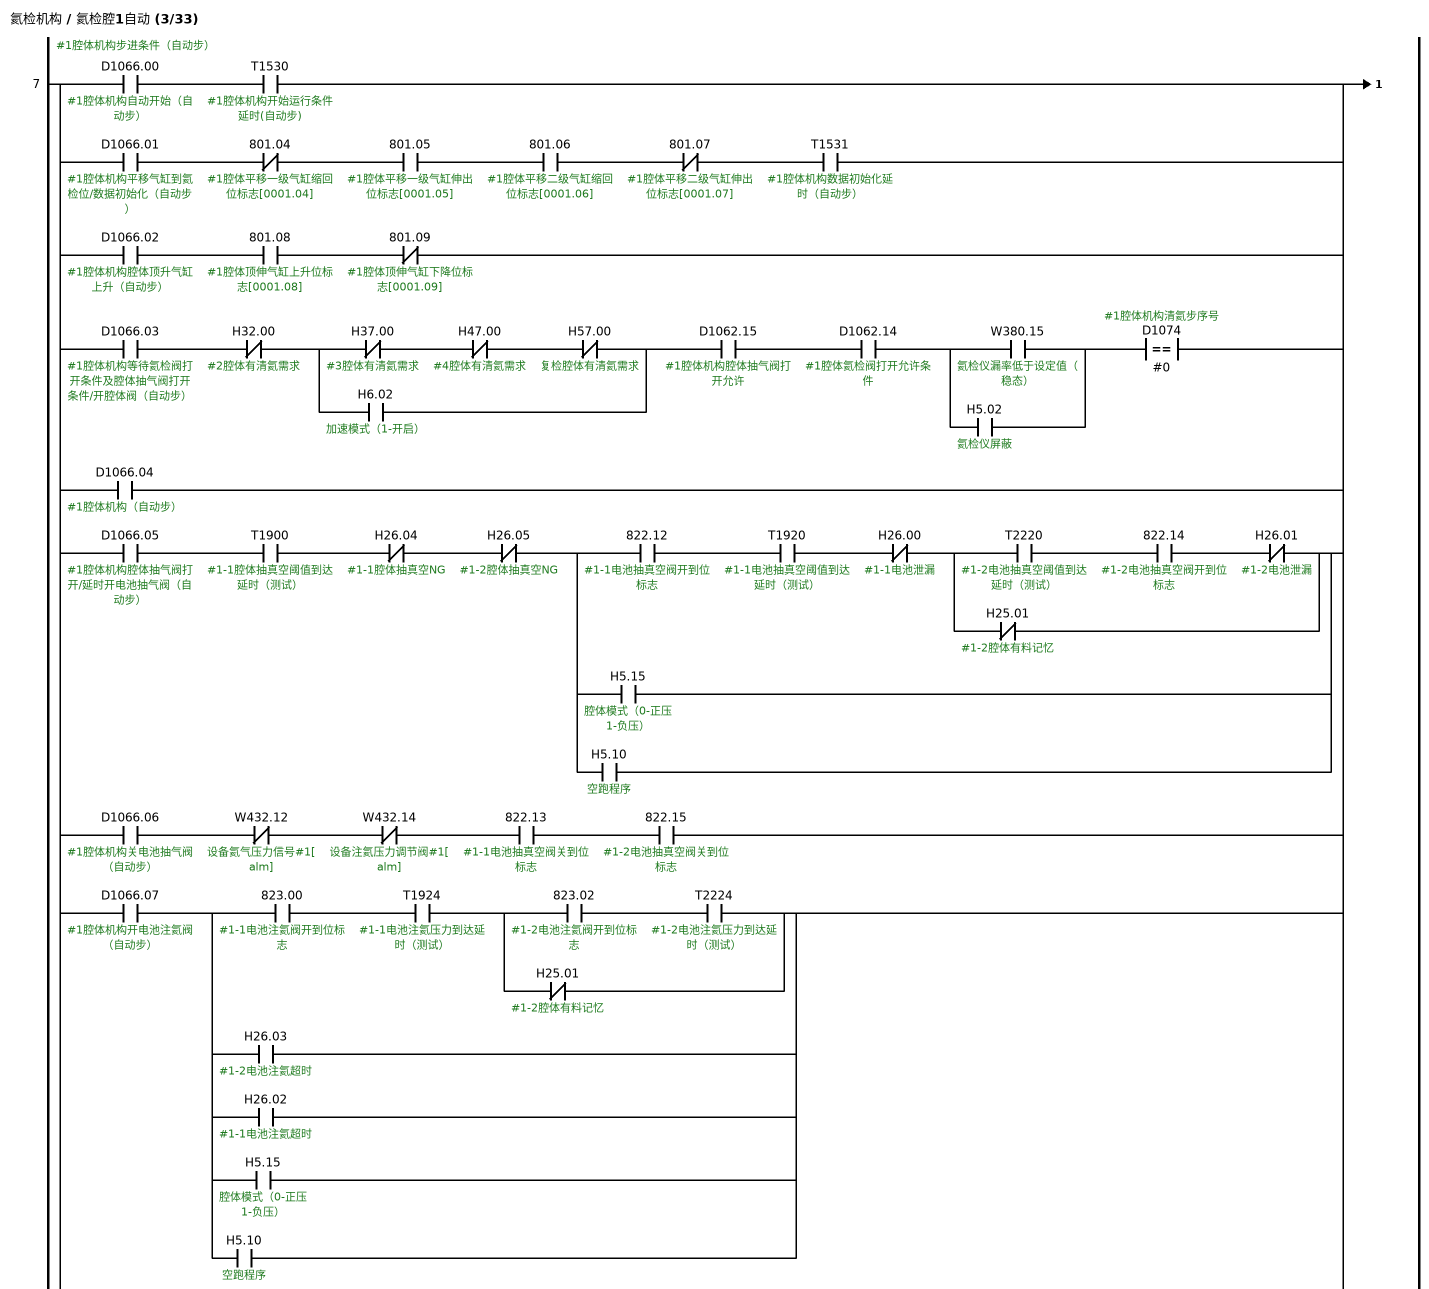

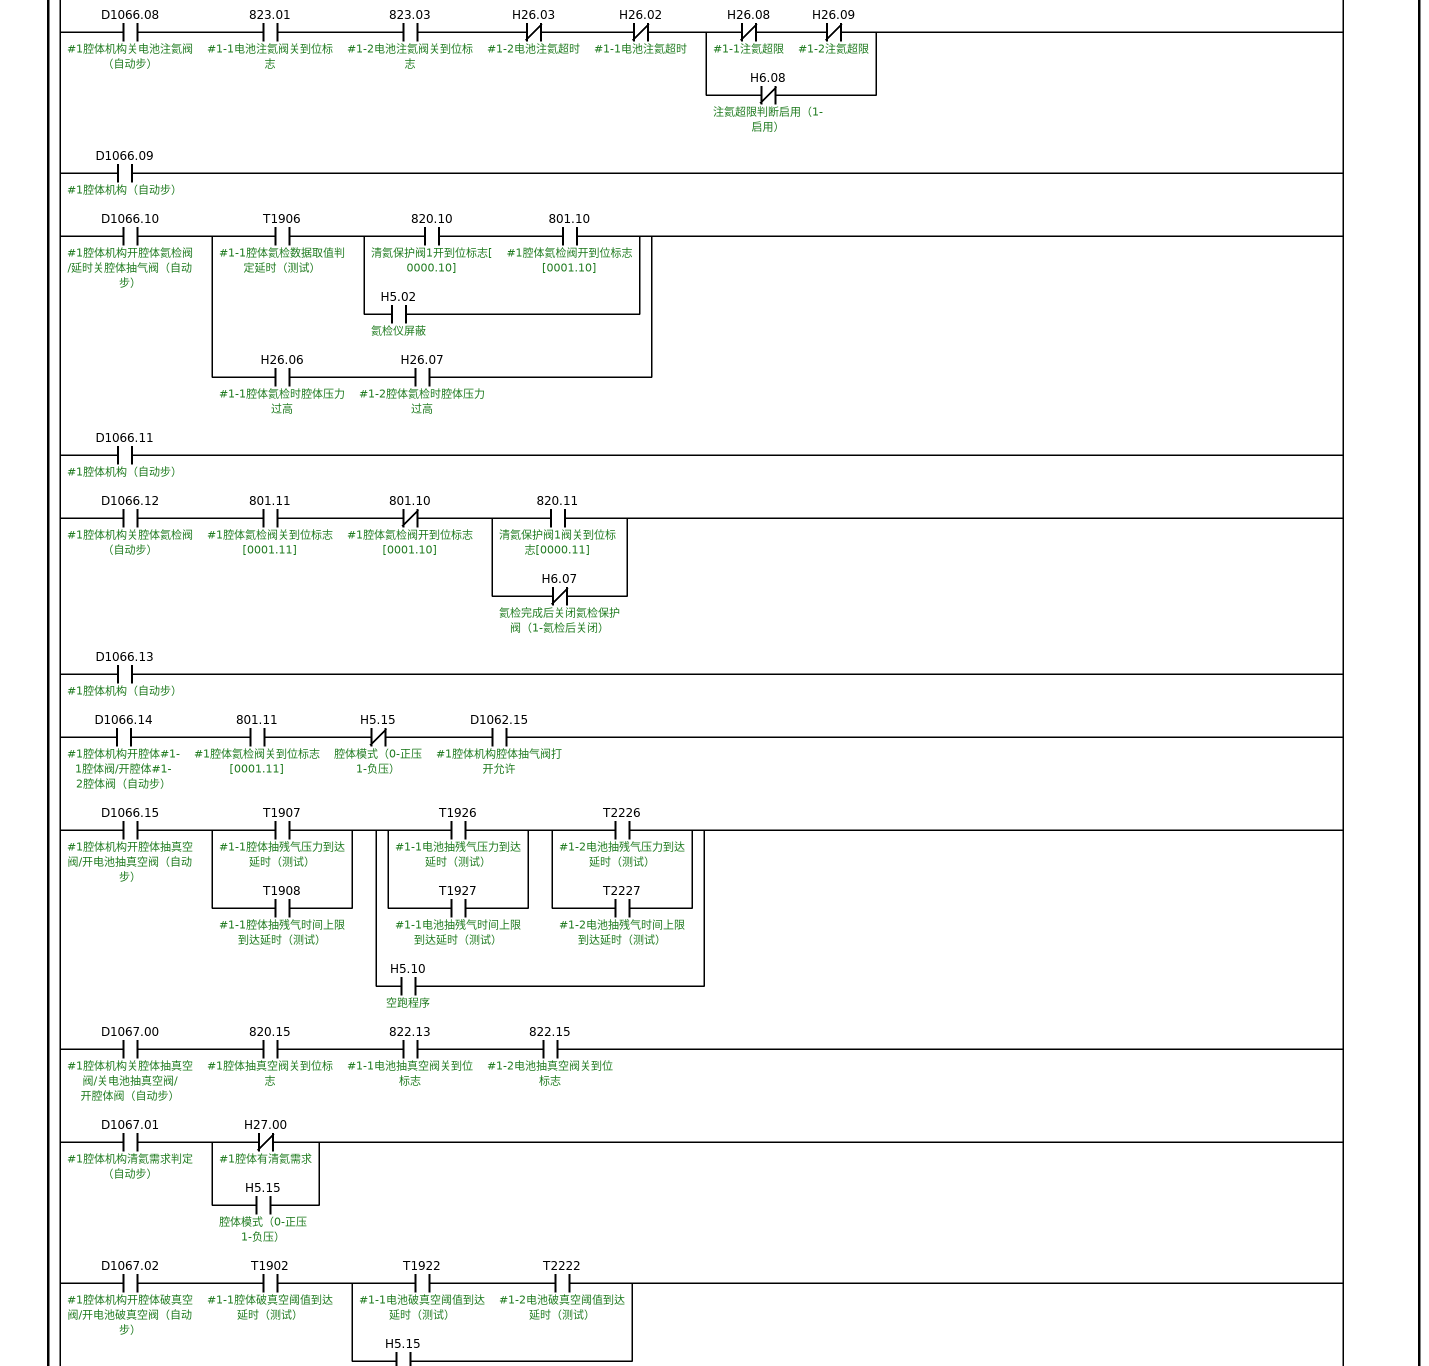

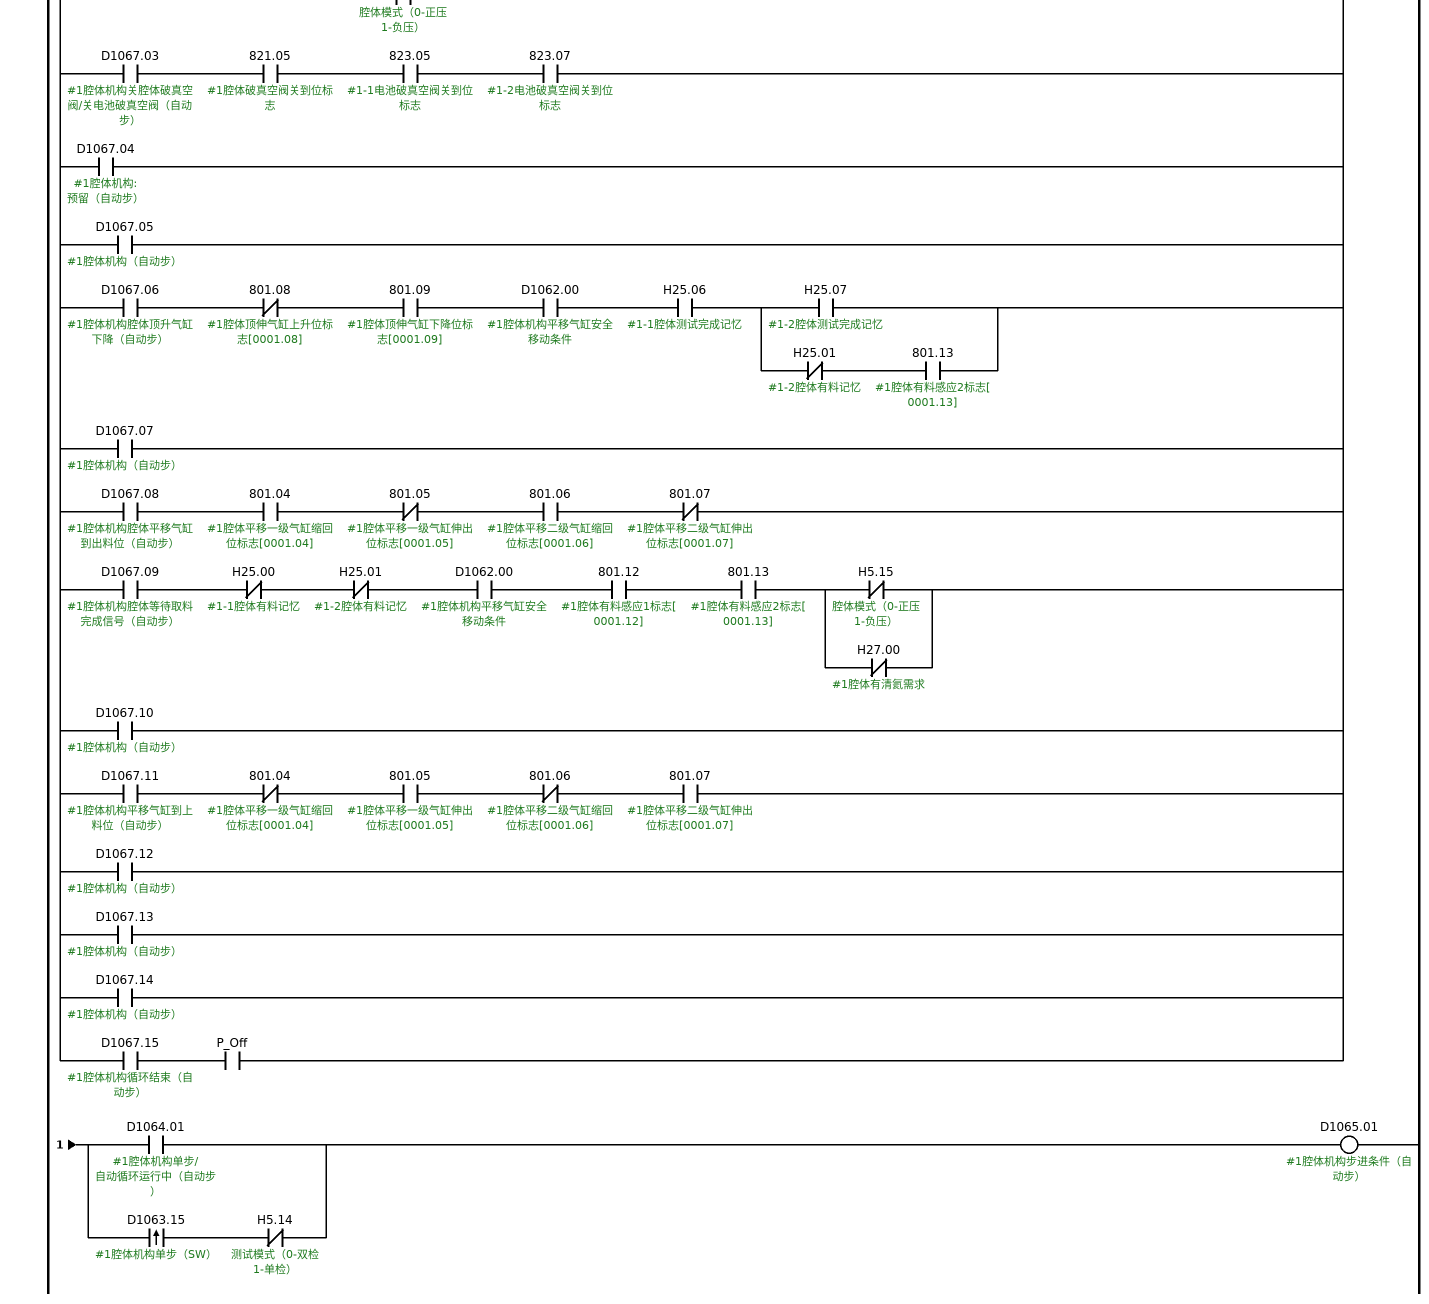
; rung 7: #1腔体机构步进条件（自动步）
LD D1066.00  ; #1腔体机构自动开始（自动步）
AND T1530  ; #1腔体机构开始运行条件延时(自动步)
LD D1066.01  ; #1腔体机构平移气缸到氦检位/数据初始化（自动步）
ANDNOT 801.04  ; #1腔体平移一级气缸缩回位标志[0001.04]
AND 801.05  ; #1腔体平移一级气缸伸出位标志[0001.05]
AND 801.06  ; #1腔体平移二级气缸缩回位标志[0001.06]
ANDNOT 801.07  ; #1腔体平移二级气缸伸出位标志[0001.07]
AND T1531  ; #1腔体机构数据初始化延时（自动步）
ORLD
LD D1066.02  ; #1腔体机构腔体顶升气缸上升（自动步）
AND 801.08  ; #1腔体顶伸气缸上升位标志[0001.08]
ANDNOT 801.09  ; #1腔体顶伸气缸下降位标志[0001.09]
ORLD
LD D1066.03  ; #1腔体机构等待氦检阀打开条件及腔体抽气阀打开条件/开腔体阀（自动步）
ANDNOT H32.00  ; #2腔体有清氦需求
LDNOT H37.00  ; #3腔体有清氦需求
ANDNOT H47.00  ; #4腔体有清氦需求
ANDNOT H57.00  ; 复检腔体有清氦需求
OR H6.02  ; 加速模式（1-开启）
ANDLD
AND D1062.15  ; #1腔体机构腔体抽气阀打开允许
AND D1062.14  ; #1腔体氦检阀打开允许条件
LD W380.15  ; 氦检仪漏率低于设定值（稳态）
OR H5.02  ; 氦检仪屏蔽
ANDLD
AND=L(301) D1074 #0  ; #1腔体机构清氦步序号
ORLD
OR D1066.04  ; #1腔体机构（自动步）
LD D1066.05  ; #1腔体机构腔体抽气阀打开/延时开电池抽气阀（自动步）
AND T1900  ; #1-1腔体抽真空阈值到达延时（测试）
ANDNOT H26.04  ; #1-1腔体抽真空NG
ANDNOT H26.05  ; #1-2腔体抽真空NG
LD 822.12  ; #1-1电池抽真空阀开到位标志
AND T1920  ; #1-1电池抽真空阈值到达延时（测试）
ANDNOT H26.00  ; #1-1电池泄漏
LD T2220  ; #1-2电池抽真空阈值到达延时（测试）
AND 822.14  ; #1-2电池抽真空阀开到位标志
ANDNOT H26.01  ; #1-2电池泄漏
ORNOT H25.01  ; #1-2腔体有料记忆
ANDLD
OR H5.15  ; 腔体模式（0-正压 1-负压）
OR H5.10  ; 空跑程序
ANDLD
ORLD
LD D1066.06  ; #1腔体机构关电池抽气阀（自动步）
ANDNOT W432.12  ; 设备氦气压力信号#1[alm]
ANDNOT W432.14  ; 设备注氦压力调节阀#1[alm]
AND 822.13  ; #1-1电池抽真空阀关到位标志
AND 822.15  ; #1-2电池抽真空阀关到位标志
ORLD
LD D1066.07  ; #1腔体机构开电池注氦阀（自动步）
LD 823.00  ; #1-1电池注氦阀开到位标志
AND T1924  ; #1-1电池注氦压力到达延时（测试）
LD 823.02  ; #1-2电池注氦阀开到位标志
AND T2224  ; #1-2电池注氦压力到达延时（测试）
ORNOT H25.01  ; #1-2腔体有料记忆
ANDLD
OR H26.03  ; #1-2电池注氦超时
OR H26.02  ; #1-1电池注氦超时
OR H5.15  ; 腔体模式（0-正压 1-负压）
OR H5.10  ; 空跑程序
ANDLD
ORLD
LD D1066.08  ; #1腔体机构关电池注氦阀（自动步）
AND 823.01  ; #1-1电池注氦阀关到位标志
AND 823.03  ; #1-2电池注氦阀关到位标志
ANDNOT H26.03  ; #1-2电池注氦超时
ANDNOT H26.02  ; #1-1电池注氦超时
LDNOT H26.08  ; #1-1注氦超限
ANDNOT H26.09  ; #1-2注氦超限
ORNOT H6.08  ; 注氦超限判断启用（1-启用）
ANDLD
ORLD
OR D1066.09  ; #1腔体机构（自动步）
LD D1066.10  ; #1腔体机构开腔体氦检阀/延时关腔体抽气阀（自动步）
LD T1906  ; #1-1腔体氦检数据取值判定延时（测试）
LD 820.10  ; 清氦保护阀1开到位标志[0000.10]
AND 801.10  ; #1腔体氦检阀开到位标志[0001.10]
OR H5.02  ; 氦检仪屏蔽
ANDLD
LD H26.06  ; #1-1腔体氦检时腔体压力过高
AND H26.07  ; #1-2腔体氦检时腔体压力过高
ORLD
ANDLD
ORLD
OR D1066.11  ; #1腔体机构（自动步）
LD D1066.12  ; #1腔体机构关腔体氦检阀（自动步）
AND 801.11  ; #1腔体氦检阀关到位标志[0001.11]
ANDNOT 801.10  ; #1腔体氦检阀开到位标志[0001.10]
LD 820.11  ; 清氦保护阀1阀关到位标志[0000.11]
ORNOT H6.07  ; 氦检完成后关闭氦检保护阀（1-氦检后关闭）
ANDLD
ORLD
OR D1066.13  ; #1腔体机构（自动步）
LD D1066.14  ; #1腔体机构开腔体#1-1腔体阀/开腔体#1-2腔体阀（自动步）
AND 801.11  ; #1腔体氦检阀关到位标志[0001.11]
ANDNOT H5.15  ; 腔体模式（0-正压 1-负压）
AND D1062.15  ; #1腔体机构腔体抽气阀打开允许
ORLD
LD D1066.15  ; #1腔体机构开腔体抽真空阀/开电池抽真空阀（自动步）
LD T1907  ; #1-1腔体抽残气压力到达延时（测试）
OR T1908  ; #1-1腔体抽残气时间上限到达延时（测试）
ANDLD
LD T1926  ; #1-1电池抽残气压力到达延时（测试）
OR T1927  ; #1-1电池抽残气时间上限到达延时（测试）
LD T2226  ; #1-2电池抽残气压力到达延时（测试）
OR T2227  ; #1-2电池抽残气时间上限到达延时（测试）
ANDLD
OR H5.10  ; 空跑程序
ANDLD
ORLD
LD D1067.00  ; #1腔体机构关腔体抽真空阀/关电池抽真空阀/开腔体阀（自动步）
AND 820.15  ; #1腔体抽真空阀关到位标志
AND 822.13  ; #1-1电池抽真空阀关到位标志
AND 822.15  ; #1-2电池抽真空阀关到位标志
ORLD
LD D1067.01  ; #1腔体机构清氦需求判定（自动步）
LDNOT H27.00  ; #1腔体有清氦需求
OR H5.15  ; 腔体模式（0-正压 1-负压）
ANDLD
ORLD
LD D1067.02  ; #1腔体机构开腔体破真空阀/开电池破真空阀（自动步）
AND T1902  ; #1-1腔体破真空阈值到达延时（测试）
LD T1922  ; #1-1电池破真空阈值到达延时（测试）
AND T2222  ; #1-2电池破真空阈值到达延时（测试）
OR H5.15  ; 腔体模式（0-正压 1-负压）
ANDLD
ORLD
LD D1067.03  ; #1腔体机构关腔体破真空阀/关电池破真空阀（自动步）
AND 821.05  ; #1腔体破真空阀关到位标志
AND 823.05  ; #1-1电池破真空阀关到位标志
AND 823.07  ; #1-2电池破真空阀关到位标志
ORLD
OR D1067.04  ; #1腔体机构:预留（自动步）
OR D1067.05  ; #1腔体机构（自动步）
LD D1067.06  ; #1腔体机构腔体顶升气缸下降（自动步）
ANDNOT 801.08  ; #1腔体顶伸气缸上升位标志[0001.08]
AND 801.09  ; #1腔体顶伸气缸下降位标志[0001.09]
AND D1062.00  ; #1腔体机构平移气缸安全移动条件
AND H25.06  ; #1-1腔体测试完成记忆
LD H25.07  ; #1-2腔体测试完成记忆
LDNOT H25.01  ; #1-2腔体有料记忆
AND 801.13  ; #1腔体有料感应2标志[0001.13]
ORLD
ANDLD
ORLD
OR D1067.07  ; #1腔体机构（自动步）
LD D1067.08  ; #1腔体机构腔体平移气缸到出料位（自动步）
AND 801.04  ; #1腔体平移一级气缸缩回位标志[0001.04]
ANDNOT 801.05  ; #1腔体平移一级气缸伸出位标志[0001.05]
AND 801.06  ; #1腔体平移二级气缸缩回位标志[0001.06]
ANDNOT 801.07  ; #1腔体平移二级气缸伸出位标志[0001.07]
ORLD
LD D1067.09  ; #1腔体机构腔体等待取料完成信号（自动步）  // 负压有清氦需求时，无需回初始位,直接跳回初始步序（D1066.00）
ANDNOT H25.00  ; #1-1腔体有料记忆
ANDNOT H25.01  ; #1-2腔体有料记忆
AND D1062.00  ; #1腔体机构平移气缸安全移动条件
AND 801.12  ; #1腔体有料感应1标志[0001.12]
AND 801.13  ; #1腔体有料感应2标志[0001.13]
LDNOT H5.15  ; 腔体模式（0-正压 1-负压）
ORNOT H27.00  ; #1腔体有清氦需求
ANDLD
ORLD
OR D1067.10  ; #1腔体机构（自动步）
LD D1067.11  ; #1腔体机构平移气缸到上料位（自动步）
ANDNOT 801.04  ; #1腔体平移一级气缸缩回位标志[0001.04]
AND 801.05  ; #1腔体平移一级气缸伸出位标志[0001.05]
ANDNOT 801.06  ; #1腔体平移二级气缸缩回位标志[0001.06]
AND 801.07  ; #1腔体平移二级气缸伸出位标志[0001.07]
ORLD
OR D1067.12  ; #1腔体机构（自动步）
OR D1067.13  ; #1腔体机构（自动步）
OR D1067.14  ; #1腔体机构（自动步）
LD D1067.15  ; #1腔体机构循环结束（自动步）
AND P_Off
ORLD
LD D1064.01  ; #1腔体机构单步/自动循环运行中（自动步）
@LD D1063.15  ; #1腔体机构单步（SW）
ANDNOT H5.14  ; 测试模式（0-双检 1-单检）
ORLD
ANDLD
OUT D1065.01  ; #1腔体机构步进条件（自动步）

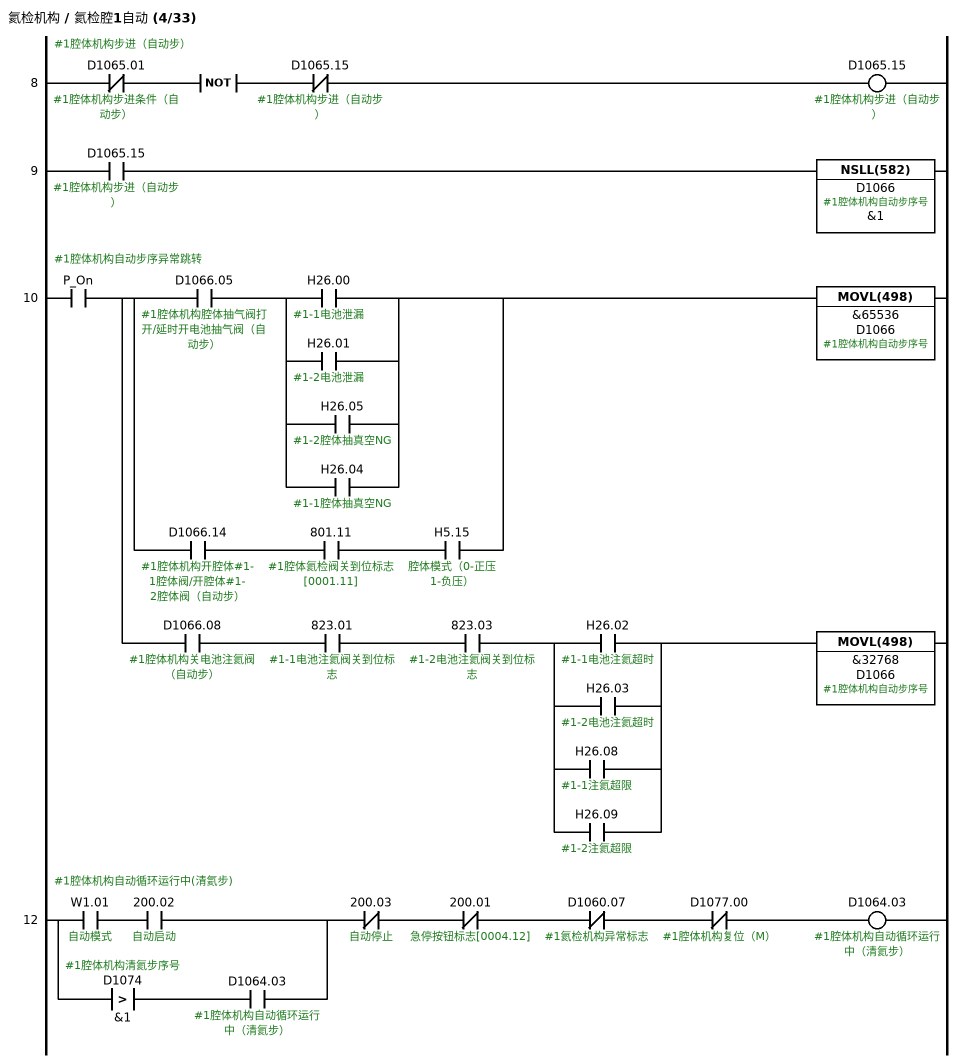
; rung 8: #1腔体机构步进（自动步）
LDNOT D1065.01  ; #1腔体机构步进条件（自动步）
NOT(520)
ANDNOT D1065.15  ; #1腔体机构步进（自动步）
OUT D1065.15  ; #1腔体机构步进（自动步）
; rung 9
LD D1065.15  ; #1腔体机构步进（自动步）
NSLL(582) D1066 &1  ; #1腔体机构自动步序号
; rung 10: #1腔体机构自动步序异常跳转
LD P_On
OUT TR0
LD D1066.05  ; #1腔体机构腔体抽气阀打开/延时开电池抽气阀（自动步）
LD H26.00  ; #1-1电池泄漏
OR H26.01  ; #1-2电池泄漏
OR H26.05  ; #1-2腔体抽真空NG
OR H26.04  ; #1-1腔体抽真空NG
ANDLD
LD D1066.14  ; #1腔体机构开腔体#1-1腔体阀/开腔体#1-2腔体阀（自动步）  // 负压模式不需要进行氦检后抽真空动作
AND 801.11  ; #1腔体氦检阀关到位标志[0001.11]
AND H5.15  ; 腔体模式（0-正压 1-负压）
ORLD
ANDLD
MOVL(498) &65536 D1066  ; #1腔体机构自动步序号  // 出现腔体抽真空NG，双电池抽真空NG，均跳转至自动步序D1067.0
LD TR0
AND D1066.08  ; #1腔体机构关电池注氦阀（自动步）
AND 823.01  ; #1-1电池注氦阀关到位标志
AND 823.03  ; #1-2电池注氦阀关到位标志
LD H26.02  ; #1-1电池注氦超时
OR H26.03  ; #1-2电池注氦超时
OR H26.08  ; #1-1注氦超限
OR H26.09  ; #1-2注氦超限
ANDLD
MOVL(498) &32768 D1066  ; #1腔体机构自动步序号  // 注氦超时需进行清氦动作（D1066.15）
; rung 11: ******************************* / 清氦步序 / *******************************
; rung 12: #1腔体机构自动循环运行中(清氦步)
LD W1.01  ; 自动模式
AND 200.02  ; 自动启动
LD>L(321) D1074 &1  ; #1腔体机构清氦步序号
AND D1064.03  ; #1腔体机构自动循环运行中（清氦步）
ORLD
ANDNOT 200.03  ; 自动停止
ANDNOT 200.01  ; 急停按钮标志[0004.12]
ANDNOT D1060.07  ; #1氦检机构异常标志
ANDNOT D1077.00  ; #1腔体机构复位（M）
OUT D1064.03  ; #1腔体机构自动循环运行中（清氦步）

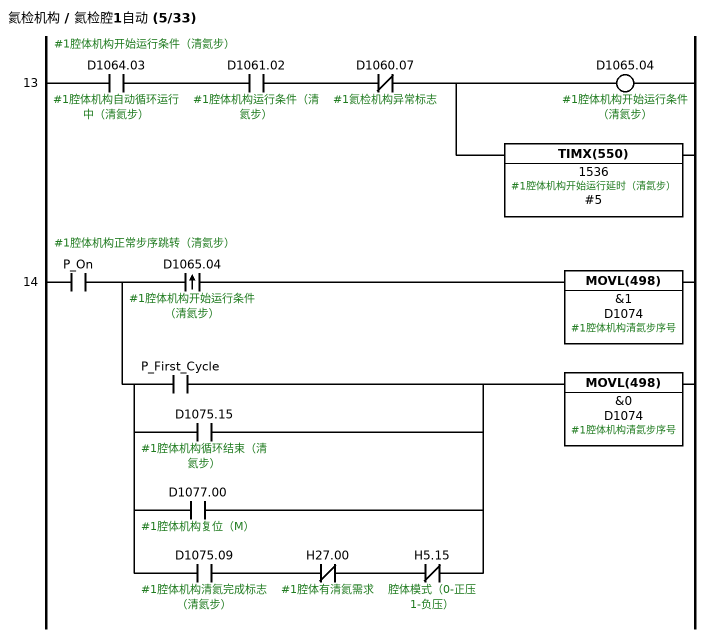
; rung 13: #1腔体机构开始运行条件（清氦步）
LD D1064.03  ; #1腔体机构自动循环运行中（清氦步）
AND D1061.02  ; #1腔体机构运行条件（清氦步）
ANDNOT D1060.07  ; #1氦检机构异常标志
OUT D1065.04  ; #1腔体机构开始运行条件（清氦步）
TIMX(550) 1536 #5  ; #1腔体机构开始运行延时（清氦步）
; rung 14: #1腔体机构正常步序跳转（清氦步）
LD P_On
OUT TR0
@AND D1065.04  ; #1腔体机构开始运行条件（清氦步）
MOVL(498) &1 D1074  ; #1腔体机构清氦步序号
LD TR0
LD P_First_Cycle
OR D1075.15  ; #1腔体机构循环结束（清氦步）
OR D1077.00  ; #1腔体机构复位（M）
LD D1075.09  ; #1腔体机构清氦完成标志（清氦步）  // 正压腔体是待料清氦，需跳转回测试步序
ANDNOT H27.00  ; #1腔体有清氦需求
ANDNOT H5.15  ; 腔体模式（0-正压 1-负压）
ORLD
ANDLD
MOVL(498) &0 D1074  ; #1腔体机构清氦步序号

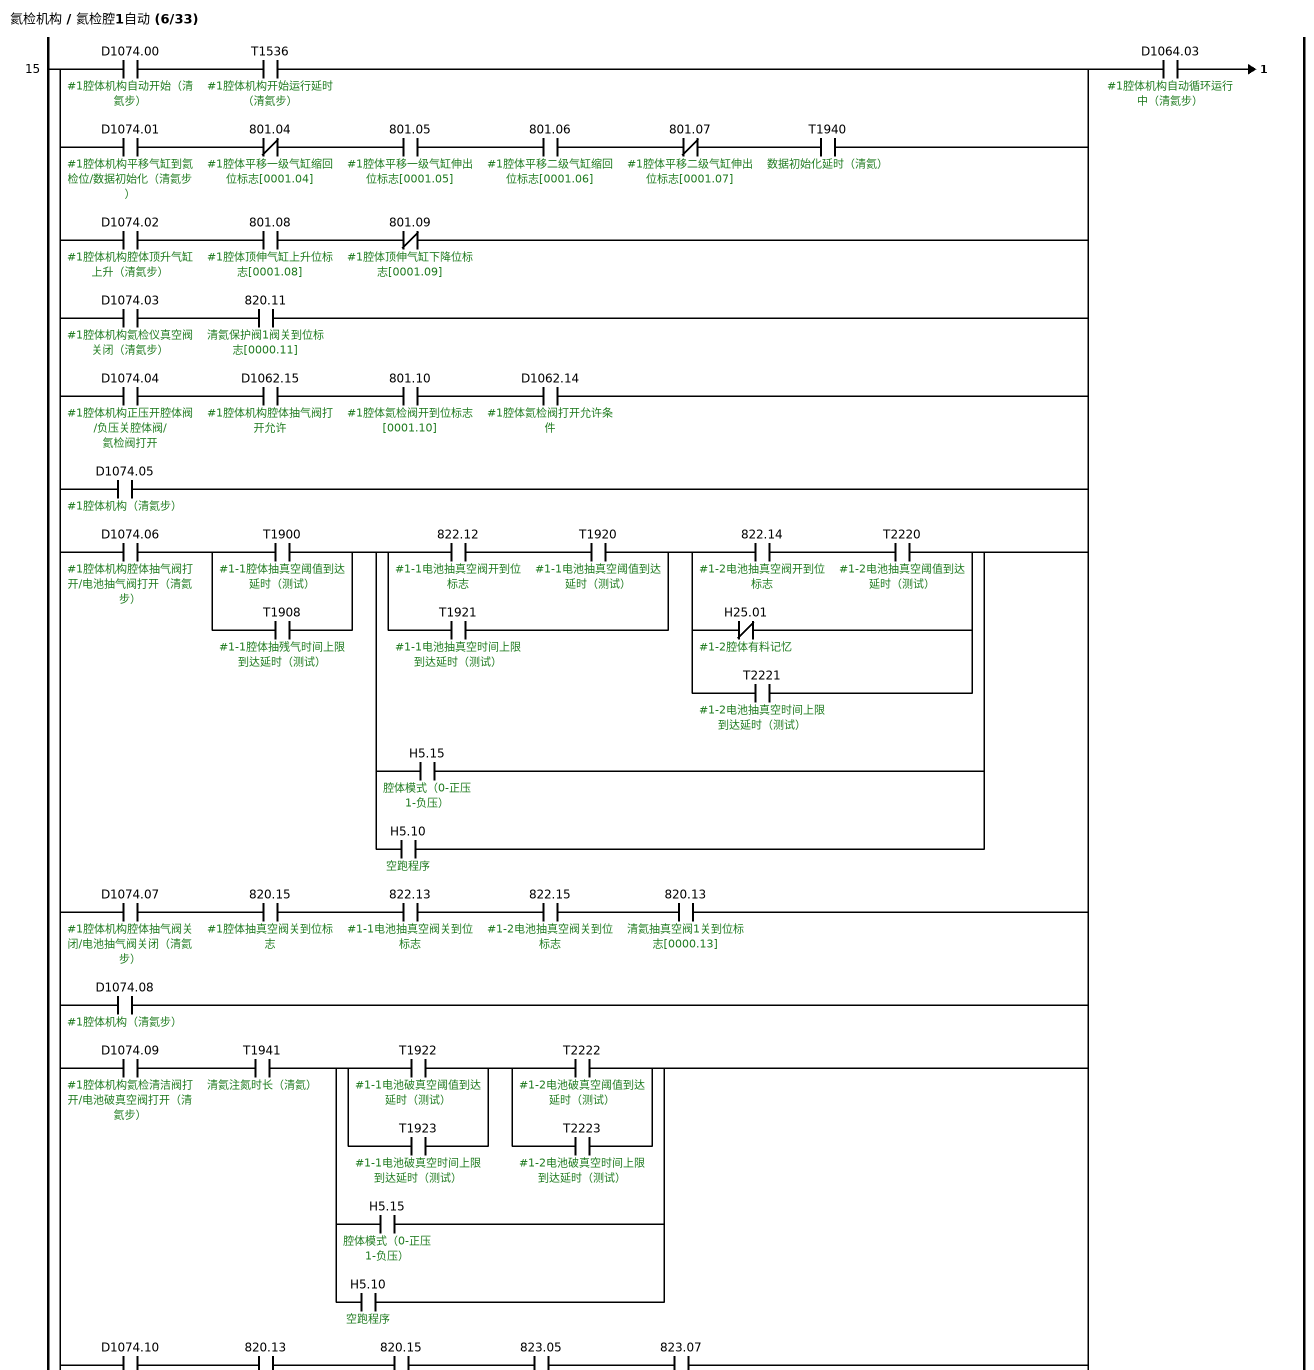

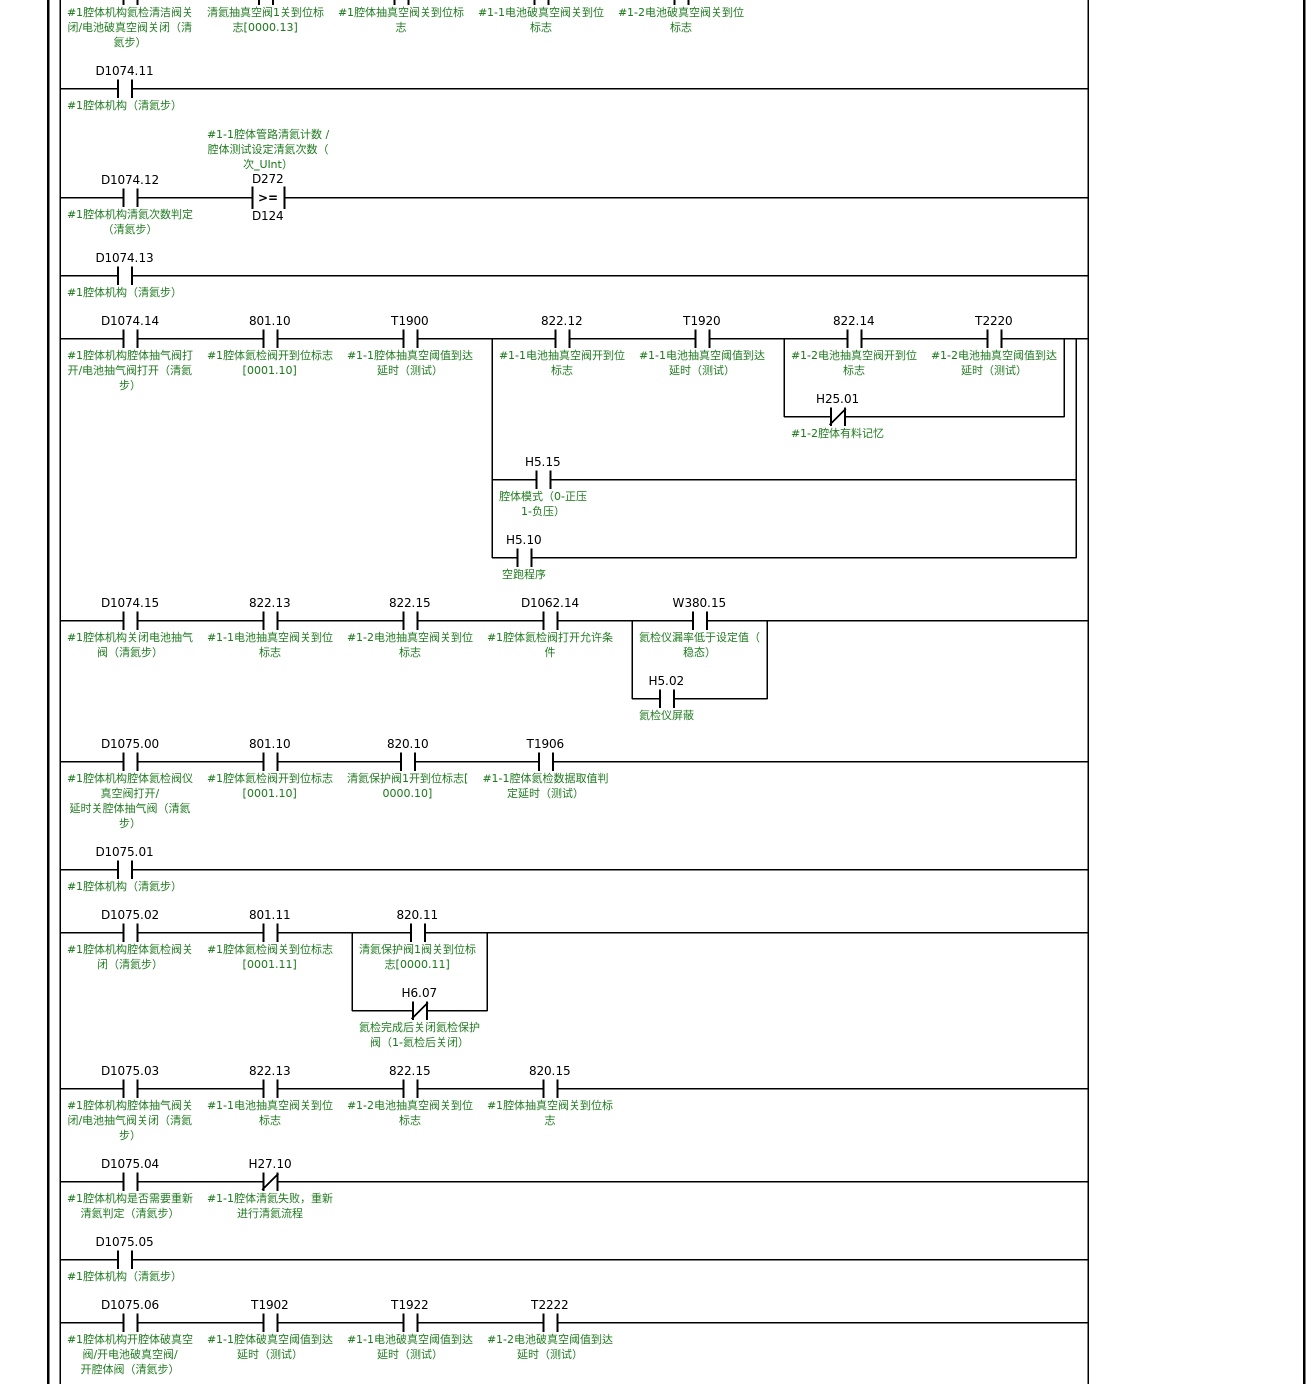

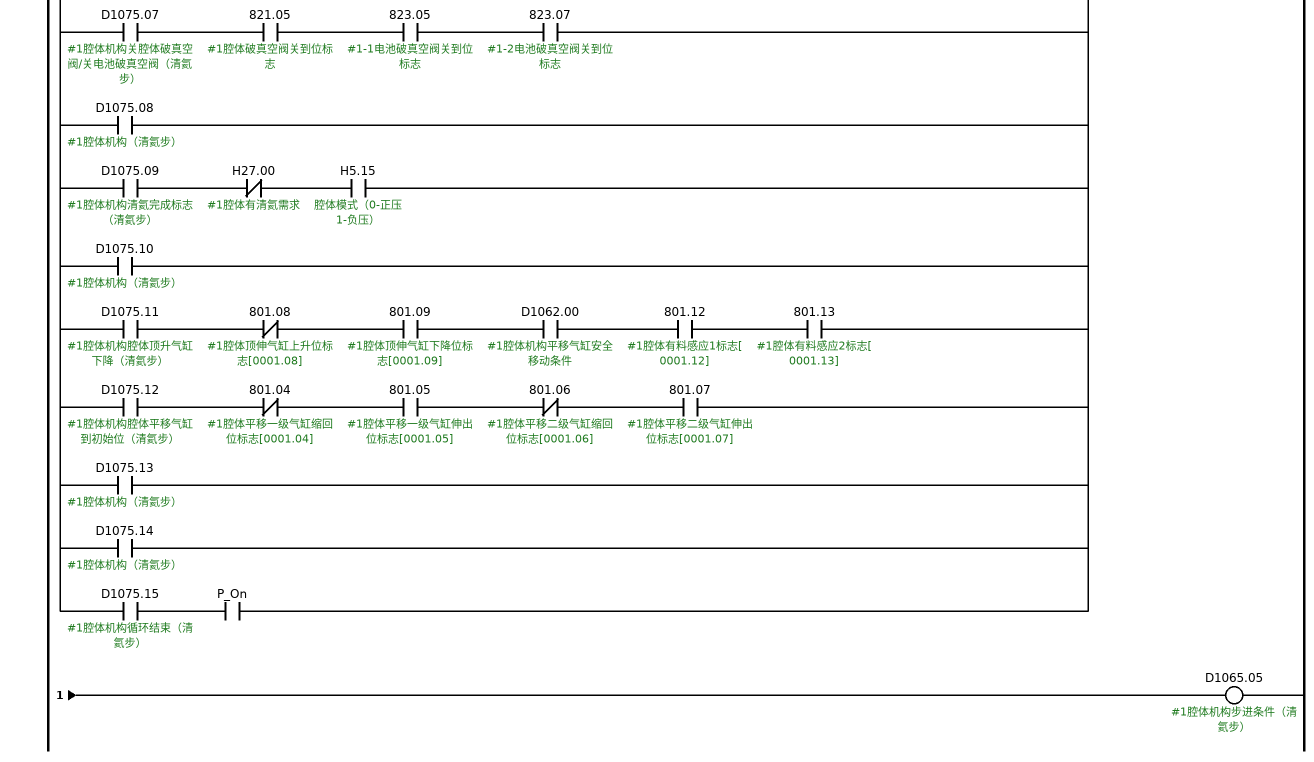
; rung 15
LD D1074.00  ; #1腔体机构自动开始（清氦步）
AND T1536  ; #1腔体机构开始运行延时（清氦步）
LD D1074.01  ; #1腔体机构平移气缸到氦检位/数据初始化（清氦步）
ANDNOT 801.04  ; #1腔体平移一级气缸缩回位标志[0001.04]
AND 801.05  ; #1腔体平移一级气缸伸出位标志[0001.05]
AND 801.06  ; #1腔体平移二级气缸缩回位标志[0001.06]
ANDNOT 801.07  ; #1腔体平移二级气缸伸出位标志[0001.07]
AND T1940  ; 数据初始化延时（清氦）
ORLD
LD D1074.02  ; #1腔体机构腔体顶升气缸上升（清氦步）
AND 801.08  ; #1腔体顶伸气缸上升位标志[0001.08]
ANDNOT 801.09  ; #1腔体顶伸气缸下降位标志[0001.09]
ORLD
LD D1074.03  ; #1腔体机构氦检仪真空阀关闭（清氦步）
AND 820.11  ; 清氦保护阀1阀关到位标志[0000.11]
ORLD
LD D1074.04  ; #1腔体机构正压开腔体阀/负压关腔体阀/氦检阀打开
AND D1062.15  ; #1腔体机构腔体抽气阀打开允许
AND 801.10  ; #1腔体氦检阀开到位标志[0001.10]
AND D1062.14  ; #1腔体氦检阀打开允许条件
ORLD
OR D1074.05  ; #1腔体机构（清氦步）
LD D1074.06  ; #1腔体机构腔体抽气阀打开/电池抽气阀打开（清氦步）
LD T1900  ; #1-1腔体抽真空阈值到达延时（测试）
OR T1908  ; #1-1腔体抽残气时间上限到达延时（测试）
ANDLD
LD 822.12  ; #1-1电池抽真空阀开到位标志
AND T1920  ; #1-1电池抽真空阈值到达延时（测试）
OR T1921  ; #1-1电池抽真空时间上限到达延时（测试）
LD 822.14  ; #1-2电池抽真空阀开到位标志
AND T2220  ; #1-2电池抽真空阈值到达延时（测试）
ORNOT H25.01  ; #1-2腔体有料记忆
OR T2221  ; #1-2电池抽真空时间上限到达延时（测试）
ANDLD
OR H5.15  ; 腔体模式（0-正压 1-负压）
OR H5.10  ; 空跑程序
ANDLD
ORLD
LD D1074.07  ; #1腔体机构腔体抽气阀关闭/电池抽气阀关闭（清氦步）
AND 820.15  ; #1腔体抽真空阀关到位标志
AND 822.13  ; #1-1电池抽真空阀关到位标志
AND 822.15  ; #1-2电池抽真空阀关到位标志
AND 820.13  ; 清氦抽真空阀1关到位标志[0000.13]
ORLD
OR D1074.08  ; #1腔体机构（清氦步）
LD D1074.09  ; #1腔体机构氦检清洁阀打开/电池破真空阀打开（清氦步）
AND T1941  ; 清氦注氮时长（清氦）
LD T1922  ; #1-1电池破真空阈值到达延时（测试）
OR T1923  ; #1-1电池破真空时间上限到达延时（测试）
LD T2222  ; #1-2电池破真空阈值到达延时（测试）
OR T2223  ; #1-2电池破真空时间上限到达延时（测试）
ANDLD
OR H5.15  ; 腔体模式（0-正压 1-负压）
OR H5.10  ; 空跑程序
ANDLD
ORLD
LD D1074.10  ; #1腔体机构氦检清洁阀关闭/电池破真空阀关闭（清氦步）
AND 820.13  ; 清氦抽真空阀1关到位标志[0000.13]
AND 820.15  ; #1腔体抽真空阀关到位标志
AND 823.05  ; #1-1电池破真空阀关到位标志
AND 823.07  ; #1-2电池破真空阀关到位标志
ORLD
OR D1074.11  ; #1腔体机构（清氦步）
LD D1074.12  ; #1腔体机构清氦次数判定（清氦步）
AND>=(325) D272 D124  ; #1-1腔体管路清氦计数, 腔体测试设定清氦次数（次_UInt）
ORLD
OR D1074.13  ; #1腔体机构（清氦步）
LD D1074.14  ; #1腔体机构腔体抽气阀打开/电池抽气阀打开（清氦步）
AND 801.10  ; #1腔体氦检阀开到位标志[0001.10]
AND T1900  ; #1-1腔体抽真空阈值到达延时（测试）
LD 822.12  ; #1-1电池抽真空阀开到位标志
AND T1920  ; #1-1电池抽真空阈值到达延时（测试）
LD 822.14  ; #1-2电池抽真空阀开到位标志
AND T2220  ; #1-2电池抽真空阈值到达延时（测试）
ORNOT H25.01  ; #1-2腔体有料记忆
ANDLD
OR H5.15  ; 腔体模式（0-正压 1-负压）
OR H5.10  ; 空跑程序
ANDLD
ORLD
LD D1074.15  ; #1腔体机构关闭电池抽气阀（清氦步）
AND 822.13  ; #1-1电池抽真空阀关到位标志
AND 822.15  ; #1-2电池抽真空阀关到位标志
AND D1062.14  ; #1腔体氦检阀打开允许条件
LD W380.15  ; 氦检仪漏率低于设定值（稳态）
OR H5.02  ; 氦检仪屏蔽
ANDLD
ORLD
LD D1075.00  ; #1腔体机构腔体氦检阀仪真空阀打开/延时关腔体抽气阀（清氦步）
AND 801.10  ; #1腔体氦检阀开到位标志[0001.10]
AND 820.10  ; 清氦保护阀1开到位标志[0000.10]
AND T1906  ; #1-1腔体氦检数据取值判定延时（测试）
ORLD
OR D1075.01  ; #1腔体机构（清氦步）
LD D1075.02  ; #1腔体机构腔体氦检阀关闭（清氦步）
AND 801.11  ; #1腔体氦检阀关到位标志[0001.11]
LD 820.11  ; 清氦保护阀1阀关到位标志[0000.11]
ORNOT H6.07  ; 氦检完成后关闭氦检保护阀（1-氦检后关闭）
ANDLD
ORLD
LD D1075.03  ; #1腔体机构腔体抽气阀关闭/电池抽气阀关闭（清氦步）
AND 822.13  ; #1-1电池抽真空阀关到位标志
AND 822.15  ; #1-2电池抽真空阀关到位标志
AND 820.15  ; #1腔体抽真空阀关到位标志
ORLD
LD D1075.04  ; #1腔体机构是否需要重新清氦判定（清氦步）
ANDNOT H27.10  ; #1-1腔体清氦失败，重新进行清氦流程  // 清氦失败，重新进行清氦
ORLD
OR D1075.05  ; #1腔体机构（清氦步）
LD D1075.06  ; #1腔体机构开腔体破真空阀/开电池破真空阀/开腔体阀（清氦步）
AND T1902  ; #1-1腔体破真空阈值到达延时（测试）
AND T1922  ; #1-1电池破真空阈值到达延时（测试）
AND T2222  ; #1-2电池破真空阈值到达延时（测试）
ORLD
LD D1075.07  ; #1腔体机构关腔体破真空阀/关电池破真空阀（清氦步）
AND 821.05  ; #1腔体破真空阀关到位标志
AND 823.05  ; #1-1电池破真空阀关到位标志
AND 823.07  ; #1-2电池破真空阀关到位标志
ORLD
OR D1075.08  ; #1腔体机构（清氦步）
LD D1075.09  ; #1腔体机构清氦完成标志（清氦步）  // 正压腔体是待料清氦，需跳转回测试步序
ANDNOT H27.00  ; #1腔体有清氦需求
AND H5.15  ; 腔体模式（0-正压 1-负压）
ORLD
OR D1075.10  ; #1腔体机构（清氦步）
LD D1075.11  ; #1腔体机构腔体顶升气缸下降（清氦步）
ANDNOT 801.08  ; #1腔体顶伸气缸上升位标志[0001.08]
AND 801.09  ; #1腔体顶伸气缸下降位标志[0001.09]
AND D1062.00  ; #1腔体机构平移气缸安全移动条件
AND 801.12  ; #1腔体有料感应1标志[0001.12]
AND 801.13  ; #1腔体有料感应2标志[0001.13]
ORLD
LD D1075.12  ; #1腔体机构腔体平移气缸到初始位（清氦步）
ANDNOT 801.04  ; #1腔体平移一级气缸缩回位标志[0001.04]
AND 801.05  ; #1腔体平移一级气缸伸出位标志[0001.05]
ANDNOT 801.06  ; #1腔体平移二级气缸缩回位标志[0001.06]
AND 801.07  ; #1腔体平移二级气缸伸出位标志[0001.07]
ORLD
OR D1075.13  ; #1腔体机构（清氦步）
OR D1075.14  ; #1腔体机构（清氦步）
LD D1075.15  ; #1腔体机构循环结束（清氦步）
AND P_On
ORLD
AND D1064.03  ; #1腔体机构自动循环运行中（清氦步）
OUT D1065.05  ; #1腔体机构步进条件（清氦步）

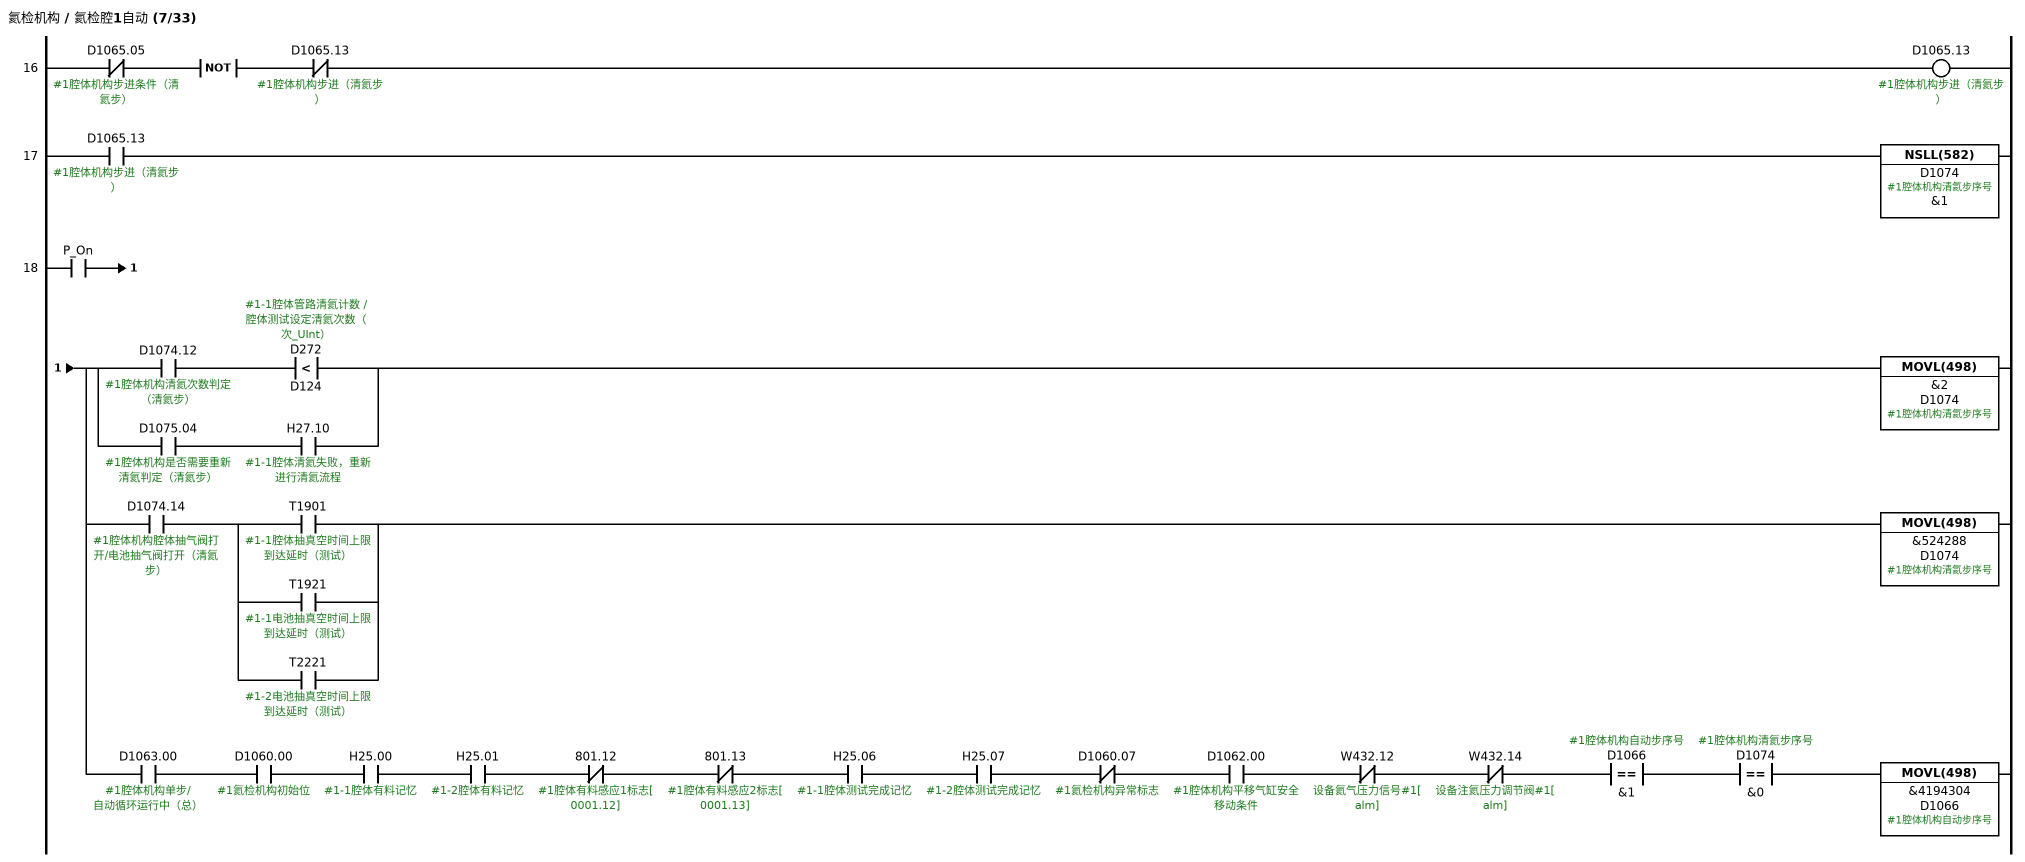
; rung 16
LDNOT D1065.05  ; #1腔体机构步进条件（清氦步）
NOT(520)
ANDNOT D1065.13  ; #1腔体机构步进（清氦步）
OUT D1065.13  ; #1腔体机构步进（清氦步）
; rung 17
LD D1065.13  ; #1腔体机构步进（清氦步）
NSLL(582) D1074 &1  ; #1腔体机构清氦步序号
; rung 18
LD P_On
OUT TR0
LD D1074.12  ; #1腔体机构清氦次数判定（清氦步）
AND<(310) D272 D124  ; #1-1腔体管路清氦计数, 腔体测试设定清氦次数（次_UInt）
LD D1075.04  ; #1腔体机构是否需要重新清氦判定（清氦步）
AND H27.10  ; #1-1腔体清氦失败，重新进行清氦流程  // 清氦失败，重新进行清氦
ORLD
ANDLD
MOVL(498) &2 D1074  ; #1腔体机构清氦步序号
LD TR0
AND D1074.14  ; #1腔体机构腔体抽气阀打开/电池抽气阀打开（清氦步）
LD T1901  ; #1-1腔体抽真空时间上限到达延时（测试）
OR T1921  ; #1-1电池抽真空时间上限到达延时（测试）
OR T2221  ; #1-2电池抽真空时间上限到达延时（测试）
ANDLD
MOVL(498) &524288 D1074  ; #1腔体机构清氦步序号  // 清氦过程腔体或电池抽气上限达到，均直接判定清氦完成，不进入氦检步序（跳转至D1075.03）
LD TR0
AND D1063.00  ; #1腔体机构单步/自动循环运行中（总）
AND D1060.00  ; #1氦检机构初始位
AND H25.00  ; #1-1腔体有料记忆
AND H25.01  ; #1-2腔体有料记忆
ANDNOT 801.12  ; #1腔体有料感应1标志[0001.12]
ANDNOT 801.13  ; #1腔体有料感应2标志[0001.13]
AND H25.06  ; #1-1腔体测试完成记忆
AND H25.07  ; #1-2腔体测试完成记忆
ANDNOT D1060.07  ; #1氦检机构异常标志
AND D1062.00  ; #1腔体机构平移气缸安全移动条件
ANDNOT W432.12  ; 设备氦气压力信号#1[alm]
ANDNOT W432.14  ; 设备注氦压力调节阀#1[alm]
AND=L(301) D1066 &1  ; #1腔体机构自动步序号
AND=L(301) D1074 &0  ; #1腔体机构清氦步序号
MOVL(498) &4194304 D1066  ; #1腔体机构自动步序号  // 带料复位时，有测试完成料则跳转到D1067.06

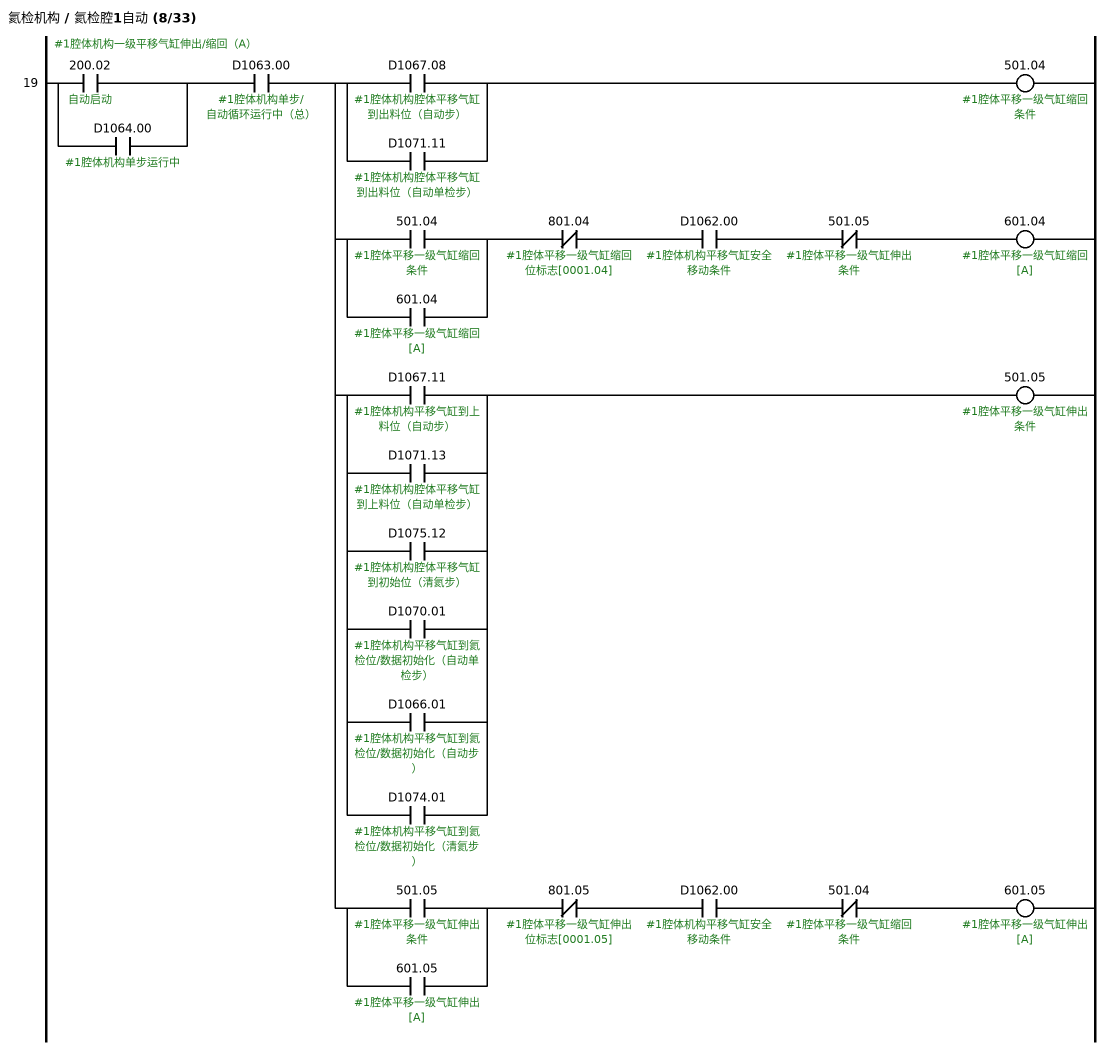
; rung 19: #1腔体机构一级平移气缸伸出/缩回（A）
LD 200.02  ; 自动启动
OR D1064.00  ; #1腔体机构单步运行中
AND D1063.00  ; #1腔体机构单步/自动循环运行中（总）
OUT TR0
LD D1067.08  ; #1腔体机构腔体平移气缸到出料位（自动步）
OR D1071.11  ; #1腔体机构腔体平移气缸到出料位（自动单检步）
ANDLD
OUT 501.04  ; #1腔体平移一级气缸缩回条件
LD TR0
LD 501.04  ; #1腔体平移一级气缸缩回条件
OR 601.04  ; #1腔体平移一级气缸缩回[A]
ANDLD
ANDNOT 801.04  ; #1腔体平移一级气缸缩回位标志[0001.04]
AND D1062.00  ; #1腔体机构平移气缸安全移动条件
ANDNOT 501.05  ; #1腔体平移一级气缸伸出条件
OUT 601.04  ; #1腔体平移一级气缸缩回[A]
LD TR0
LD D1067.11  ; #1腔体机构平移气缸到上料位（自动步）
OR D1071.13  ; #1腔体机构腔体平移气缸到上料位（自动单检步）
OR D1075.12  ; #1腔体机构腔体平移气缸到初始位（清氦步）
OR D1070.01  ; #1腔体机构平移气缸到氦检位/数据初始化（自动单检步）
OR D1066.01  ; #1腔体机构平移气缸到氦检位/数据初始化（自动步）
OR D1074.01  ; #1腔体机构平移气缸到氦检位/数据初始化（清氦步）
ANDLD
OUT 501.05  ; #1腔体平移一级气缸伸出条件
LD TR0
LD 501.05  ; #1腔体平移一级气缸伸出条件
OR 601.05  ; #1腔体平移一级气缸伸出[A]
ANDLD
ANDNOT 801.05  ; #1腔体平移一级气缸伸出位标志[0001.05]
AND D1062.00  ; #1腔体机构平移气缸安全移动条件
ANDNOT 501.04  ; #1腔体平移一级气缸缩回条件
OUT 601.05  ; #1腔体平移一级气缸伸出[A]

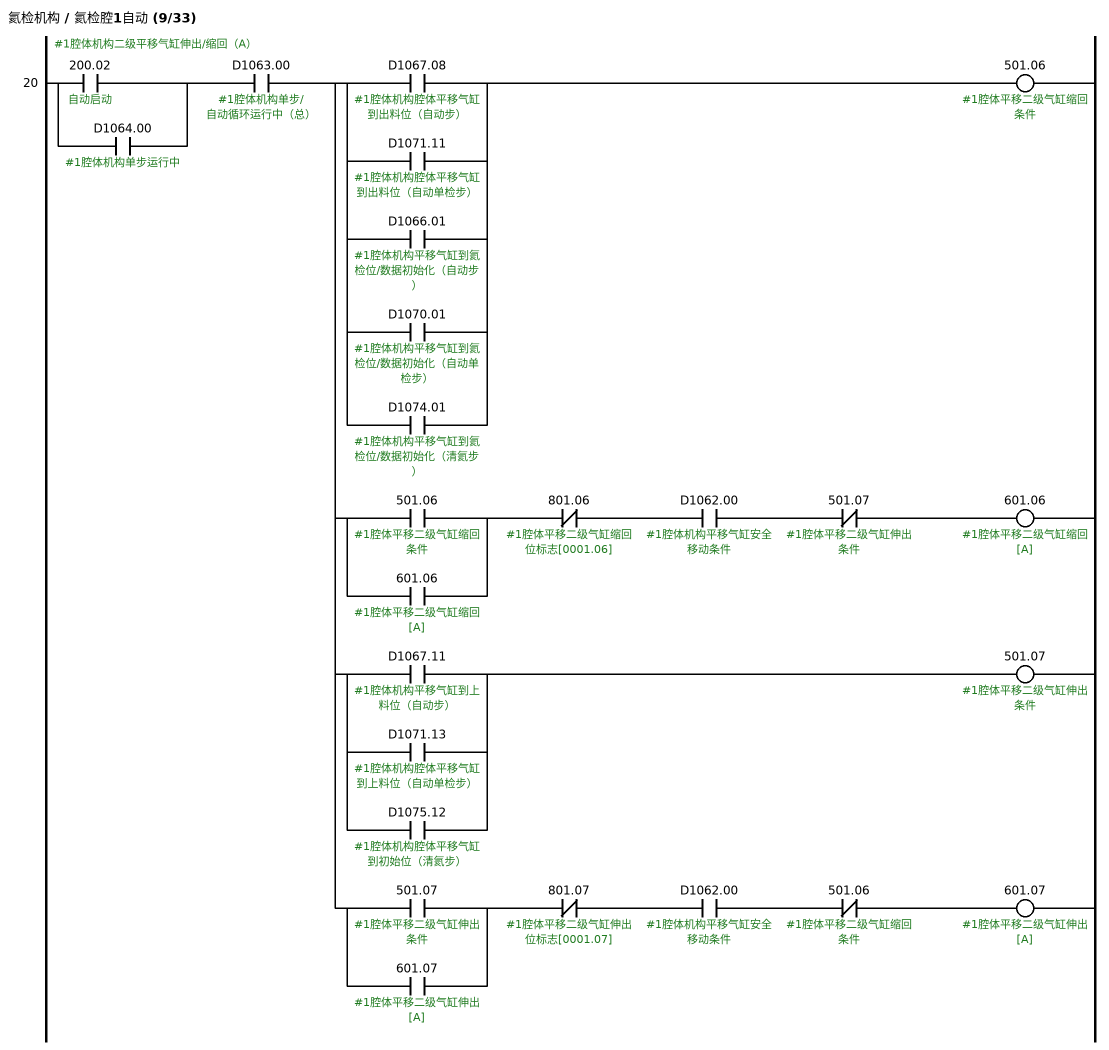
; rung 20: #1腔体机构二级平移气缸伸出/缩回（A）
LD 200.02  ; 自动启动
OR D1064.00  ; #1腔体机构单步运行中
AND D1063.00  ; #1腔体机构单步/自动循环运行中（总）
OUT TR0
LD D1067.08  ; #1腔体机构腔体平移气缸到出料位（自动步）
OR D1071.11  ; #1腔体机构腔体平移气缸到出料位（自动单检步）
OR D1066.01  ; #1腔体机构平移气缸到氦检位/数据初始化（自动步）
OR D1070.01  ; #1腔体机构平移气缸到氦检位/数据初始化（自动单检步）
OR D1074.01  ; #1腔体机构平移气缸到氦检位/数据初始化（清氦步）
ANDLD
OUT 501.06  ; #1腔体平移二级气缸缩回条件
LD TR0
LD 501.06  ; #1腔体平移二级气缸缩回条件
OR 601.06  ; #1腔体平移二级气缸缩回[A]
ANDLD
ANDNOT 801.06  ; #1腔体平移二级气缸缩回位标志[0001.06]
AND D1062.00  ; #1腔体机构平移气缸安全移动条件
ANDNOT 501.07  ; #1腔体平移二级气缸伸出条件
OUT 601.06  ; #1腔体平移二级气缸缩回[A]
LD TR0
LD D1067.11  ; #1腔体机构平移气缸到上料位（自动步）
OR D1071.13  ; #1腔体机构腔体平移气缸到上料位（自动单检步）
OR D1075.12  ; #1腔体机构腔体平移气缸到初始位（清氦步）
ANDLD
OUT 501.07  ; #1腔体平移二级气缸伸出条件
LD TR0
LD 501.07  ; #1腔体平移二级气缸伸出条件
OR 601.07  ; #1腔体平移二级气缸伸出[A]
ANDLD
ANDNOT 801.07  ; #1腔体平移二级气缸伸出位标志[0001.07]
AND D1062.00  ; #1腔体机构平移气缸安全移动条件
ANDNOT 501.06  ; #1腔体平移二级气缸缩回条件
OUT 601.07  ; #1腔体平移二级气缸伸出[A]

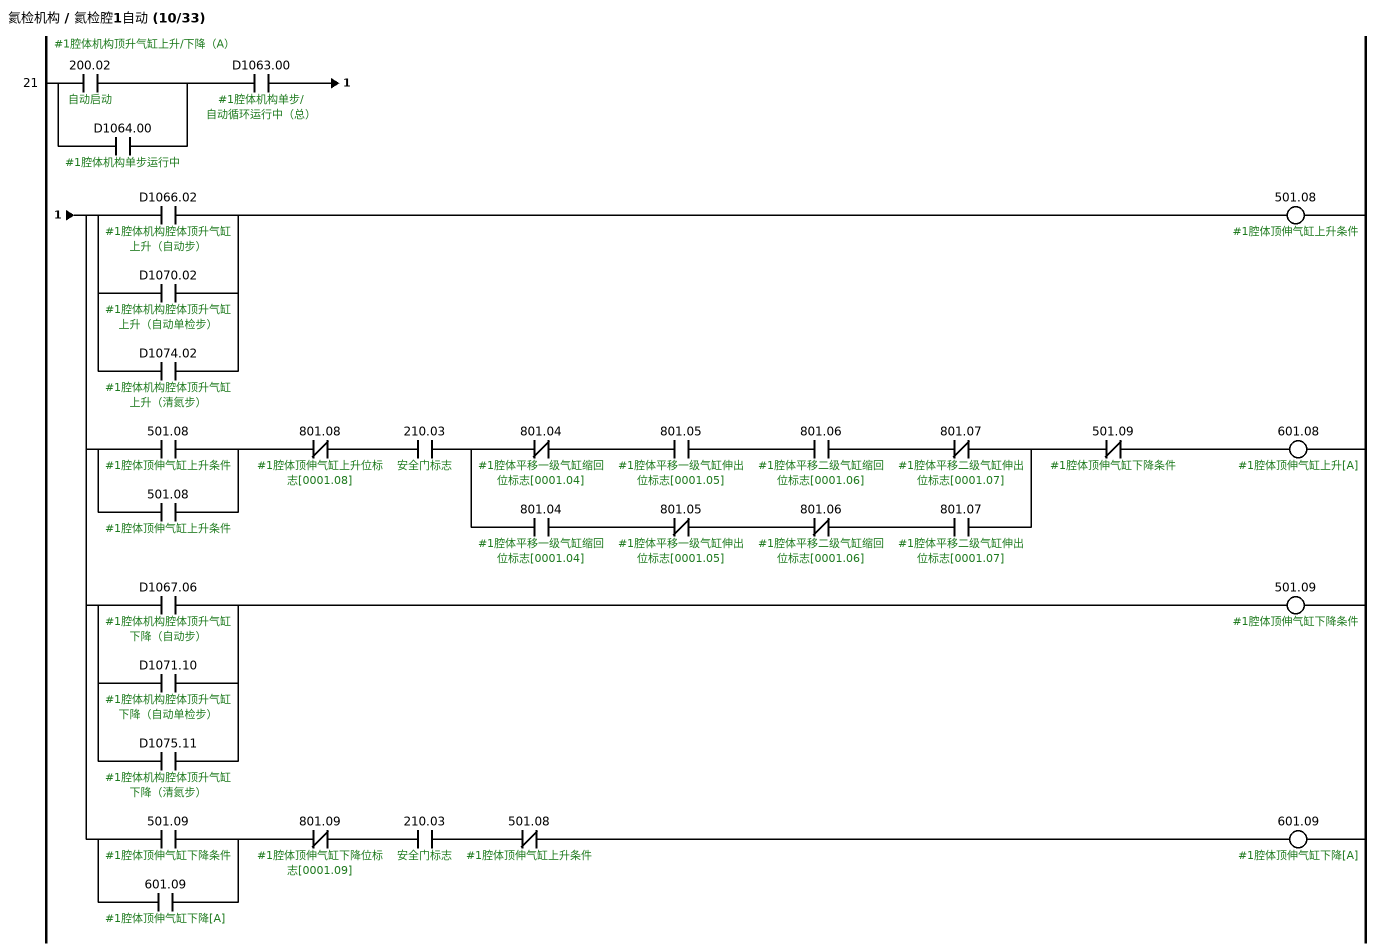
; rung 21: #1腔体机构顶升气缸上升/下降（A）
LD 200.02  ; 自动启动
OR D1064.00  ; #1腔体机构单步运行中
AND D1063.00  ; #1腔体机构单步/自动循环运行中（总）
OUT TR0
LD D1066.02  ; #1腔体机构腔体顶升气缸上升（自动步）
OR D1070.02  ; #1腔体机构腔体顶升气缸上升（自动单检步）
OR D1074.02  ; #1腔体机构腔体顶升气缸上升（清氦步）
ANDLD
OUT 501.08  ; #1腔体顶伸气缸上升条件
LD TR0
LD 501.08  ; #1腔体顶伸气缸上升条件
OR 501.08  ; #1腔体顶伸气缸上升条件
ANDLD
ANDNOT 801.08  ; #1腔体顶伸气缸上升位标志[0001.08]
AND 210.03  ; 安全门标志
LDNOT 801.04  ; #1腔体平移一级气缸缩回位标志[0001.04]
AND 801.05  ; #1腔体平移一级气缸伸出位标志[0001.05]
AND 801.06  ; #1腔体平移二级气缸缩回位标志[0001.06]
ANDNOT 801.07  ; #1腔体平移二级气缸伸出位标志[0001.07]
LD 801.04  ; #1腔体平移一级气缸缩回位标志[0001.04]
ANDNOT 801.05  ; #1腔体平移一级气缸伸出位标志[0001.05]
ANDNOT 801.06  ; #1腔体平移二级气缸缩回位标志[0001.06]
AND 801.07  ; #1腔体平移二级气缸伸出位标志[0001.07]
ORLD
ANDLD
ANDNOT 501.09  ; #1腔体顶伸气缸下降条件
OUT 601.08  ; #1腔体顶伸气缸上升[A]
LD TR0
LD D1067.06  ; #1腔体机构腔体顶升气缸下降（自动步）
OR D1071.10  ; #1腔体机构腔体顶升气缸下降（自动单检步）
OR D1075.11  ; #1腔体机构腔体顶升气缸下降（清氦步）
ANDLD
OUT 501.09  ; #1腔体顶伸气缸下降条件
LD TR0
LD 501.09  ; #1腔体顶伸气缸下降条件
OR 601.09  ; #1腔体顶伸气缸下降[A]
ANDLD
ANDNOT 801.09  ; #1腔体顶伸气缸下降位标志[0001.09]
AND 210.03  ; 安全门标志
ANDNOT 501.08  ; #1腔体顶伸气缸上升条件
OUT 601.09  ; #1腔体顶伸气缸下降[A]

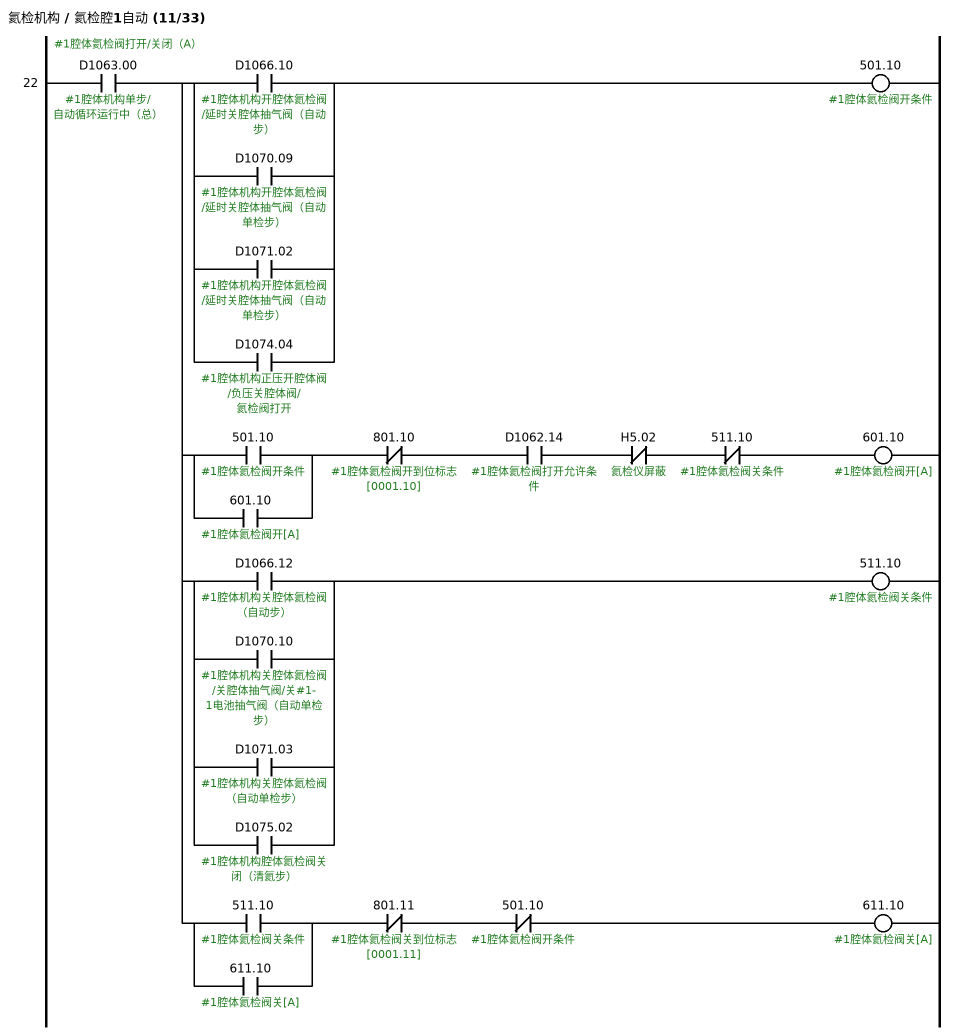
; rung 22: #1腔体氦检阀打开/关闭（A）
LD D1063.00  ; #1腔体机构单步/自动循环运行中（总）
OUT TR0
LD D1066.10  ; #1腔体机构开腔体氦检阀/延时关腔体抽气阀（自动步）
OR D1070.09  ; #1腔体机构开腔体氦检阀/延时关腔体抽气阀（自动单检步）
OR D1071.02  ; #1腔体机构开腔体氦检阀/延时关腔体抽气阀（自动单检步）
OR D1074.04  ; #1腔体机构正压开腔体阀/负压关腔体阀/氦检阀打开
ANDLD
OUT 501.10  ; #1腔体氦检阀开条件
LD TR0
LD 501.10  ; #1腔体氦检阀开条件
OR 601.10  ; #1腔体氦检阀开[A]
ANDLD
ANDNOT 801.10  ; #1腔体氦检阀开到位标志[0001.10]
AND D1062.14  ; #1腔体氦检阀打开允许条件
ANDNOT H5.02  ; 氦检仪屏蔽
ANDNOT 511.10  ; #1腔体氦检阀关条件
OUT 601.10  ; #1腔体氦检阀开[A]
LD TR0
LD D1066.12  ; #1腔体机构关腔体氦检阀（自动步）
OR D1070.10  ; #1腔体机构关腔体氦检阀/关腔体抽气阀/关#1-1电池抽气阀（自动单检步）
OR D1071.03  ; #1腔体机构关腔体氦检阀（自动单检步）
OR D1075.02  ; #1腔体机构腔体氦检阀关闭（清氦步）
ANDLD
OUT 511.10  ; #1腔体氦检阀关条件
LD TR0
LD 511.10  ; #1腔体氦检阀关条件
OR 611.10  ; #1腔体氦检阀关[A]
ANDLD
ANDNOT 801.11  ; #1腔体氦检阀关到位标志[0001.11]
ANDNOT 501.10  ; #1腔体氦检阀开条件
OUT 611.10  ; #1腔体氦检阀关[A]

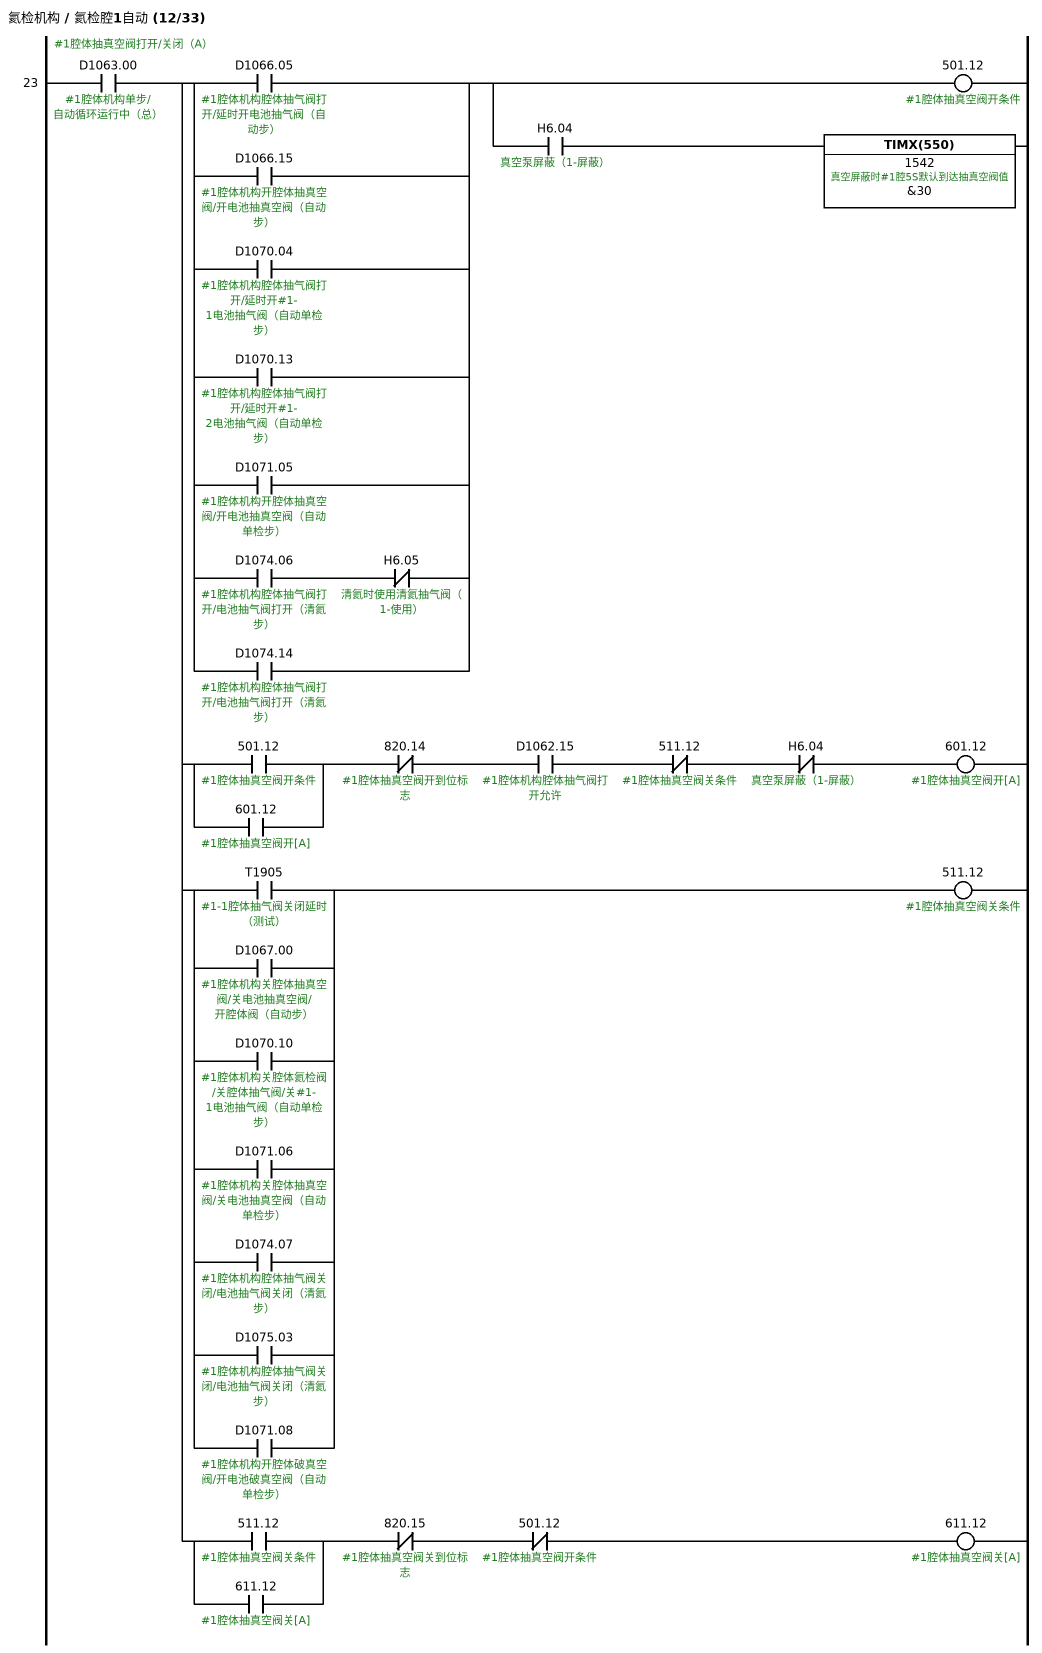
; rung 23: #1腔体抽真空阀打开/关闭（A）
LD D1063.00  ; #1腔体机构单步/自动循环运行中（总）
OUT TR0
LD D1066.05  ; #1腔体机构腔体抽气阀打开/延时开电池抽气阀（自动步）
OR D1066.15  ; #1腔体机构开腔体抽真空阀/开电池抽真空阀（自动步）
OR D1070.04  ; #1腔体机构腔体抽气阀打开/延时开#1-1电池抽气阀（自动单检步）
OR D1070.13  ; #1腔体机构腔体抽气阀打开/延时开#1-2电池抽气阀（自动单检步）
OR D1071.05  ; #1腔体机构开腔体抽真空阀/开电池抽真空阀（自动单检步）
LD D1074.06  ; #1腔体机构腔体抽气阀打开/电池抽气阀打开（清氦步）
ANDNOT H6.05  ; 清氦时使用清氦抽气阀（1-使用）
ORLD
OR D1074.14  ; #1腔体机构腔体抽气阀打开/电池抽气阀打开（清氦步）
ANDLD
OUT 501.12  ; #1腔体抽真空阀开条件
AND H6.04  ; 真空泵屏蔽（1-屏蔽）
TIMX(550) 1542 &30  ; 真空屏蔽时#1腔5S默认到达抽真空阀值
LD TR0
LD 501.12  ; #1腔体抽真空阀开条件
OR 601.12  ; #1腔体抽真空阀开[A]
ANDLD
ANDNOT 820.14  ; #1腔体抽真空阀开到位标志
AND D1062.15  ; #1腔体机构腔体抽气阀打开允许
ANDNOT 511.12  ; #1腔体抽真空阀关条件
ANDNOT H6.04  ; 真空泵屏蔽（1-屏蔽）
OUT 601.12  ; #1腔体抽真空阀开[A]
LD TR0
LD T1905  ; #1-1腔体抽气阀关闭延时（测试）
OR D1067.00  ; #1腔体机构关腔体抽真空阀/关电池抽真空阀/开腔体阀（自动步）
OR D1070.10  ; #1腔体机构关腔体氦检阀/关腔体抽气阀/关#1-1电池抽气阀（自动单检步）
OR D1071.06  ; #1腔体机构关腔体抽真空阀/关电池抽真空阀（自动单检步）
OR D1074.07  ; #1腔体机构腔体抽气阀关闭/电池抽气阀关闭（清氦步）
OR D1075.03  ; #1腔体机构腔体抽气阀关闭/电池抽气阀关闭（清氦步）
OR D1071.08  ; #1腔体机构开腔体破真空阀/开电池破真空阀（自动单检步）
ANDLD
OUT 511.12  ; #1腔体抽真空阀关条件
LD TR0
LD 511.12  ; #1腔体抽真空阀关条件
OR 611.12  ; #1腔体抽真空阀关[A]
ANDLD
ANDNOT 820.15  ; #1腔体抽真空阀关到位标志
ANDNOT 501.12  ; #1腔体抽真空阀开条件
OUT 611.12  ; #1腔体抽真空阀关[A]

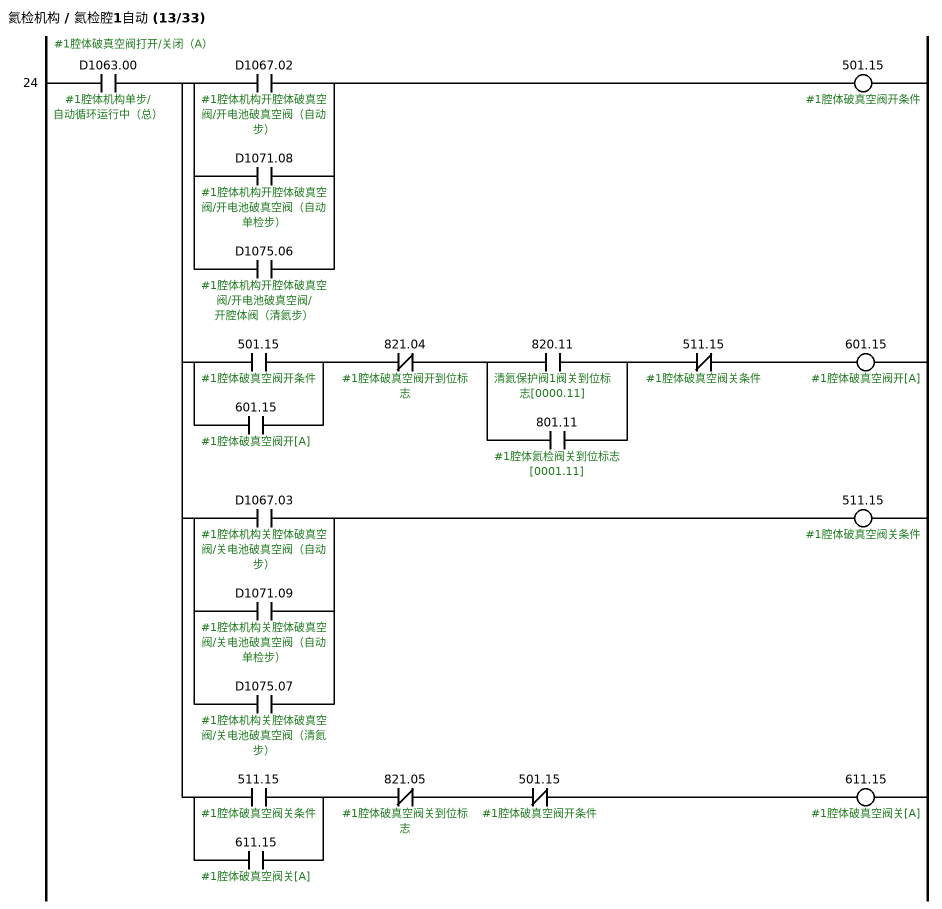
; rung 24: #1腔体破真空阀打开/关闭（A）
LD D1063.00  ; #1腔体机构单步/自动循环运行中（总）
OUT TR0
LD D1067.02  ; #1腔体机构开腔体破真空阀/开电池破真空阀（自动步）
OR D1071.08  ; #1腔体机构开腔体破真空阀/开电池破真空阀（自动单检步）
OR D1075.06  ; #1腔体机构开腔体破真空阀/开电池破真空阀/开腔体阀（清氦步）
ANDLD
OUT 501.15  ; #1腔体破真空阀开条件
LD TR0
LD 501.15  ; #1腔体破真空阀开条件
OR 601.15  ; #1腔体破真空阀开[A]
ANDLD
ANDNOT 821.04  ; #1腔体破真空阀开到位标志
LD 820.11  ; 清氦保护阀1阀关到位标志[0000.11]
OR 801.11  ; #1腔体氦检阀关到位标志[0001.11]
ANDLD
ANDNOT 511.15  ; #1腔体破真空阀关条件
OUT 601.15  ; #1腔体破真空阀开[A]
LD TR0
LD D1067.03  ; #1腔体机构关腔体破真空阀/关电池破真空阀（自动步）
OR D1071.09  ; #1腔体机构关腔体破真空阀/关电池破真空阀（自动单检步）
OR D1075.07  ; #1腔体机构关腔体破真空阀/关电池破真空阀（清氦步）
ANDLD
OUT 511.15  ; #1腔体破真空阀关条件
LD TR0
LD 511.15  ; #1腔体破真空阀关条件
OR 611.15  ; #1腔体破真空阀关[A]
ANDLD
ANDNOT 821.05  ; #1腔体破真空阀关到位标志
ANDNOT 501.15  ; #1腔体破真空阀开条件
OUT 611.15  ; #1腔体破真空阀关[A]

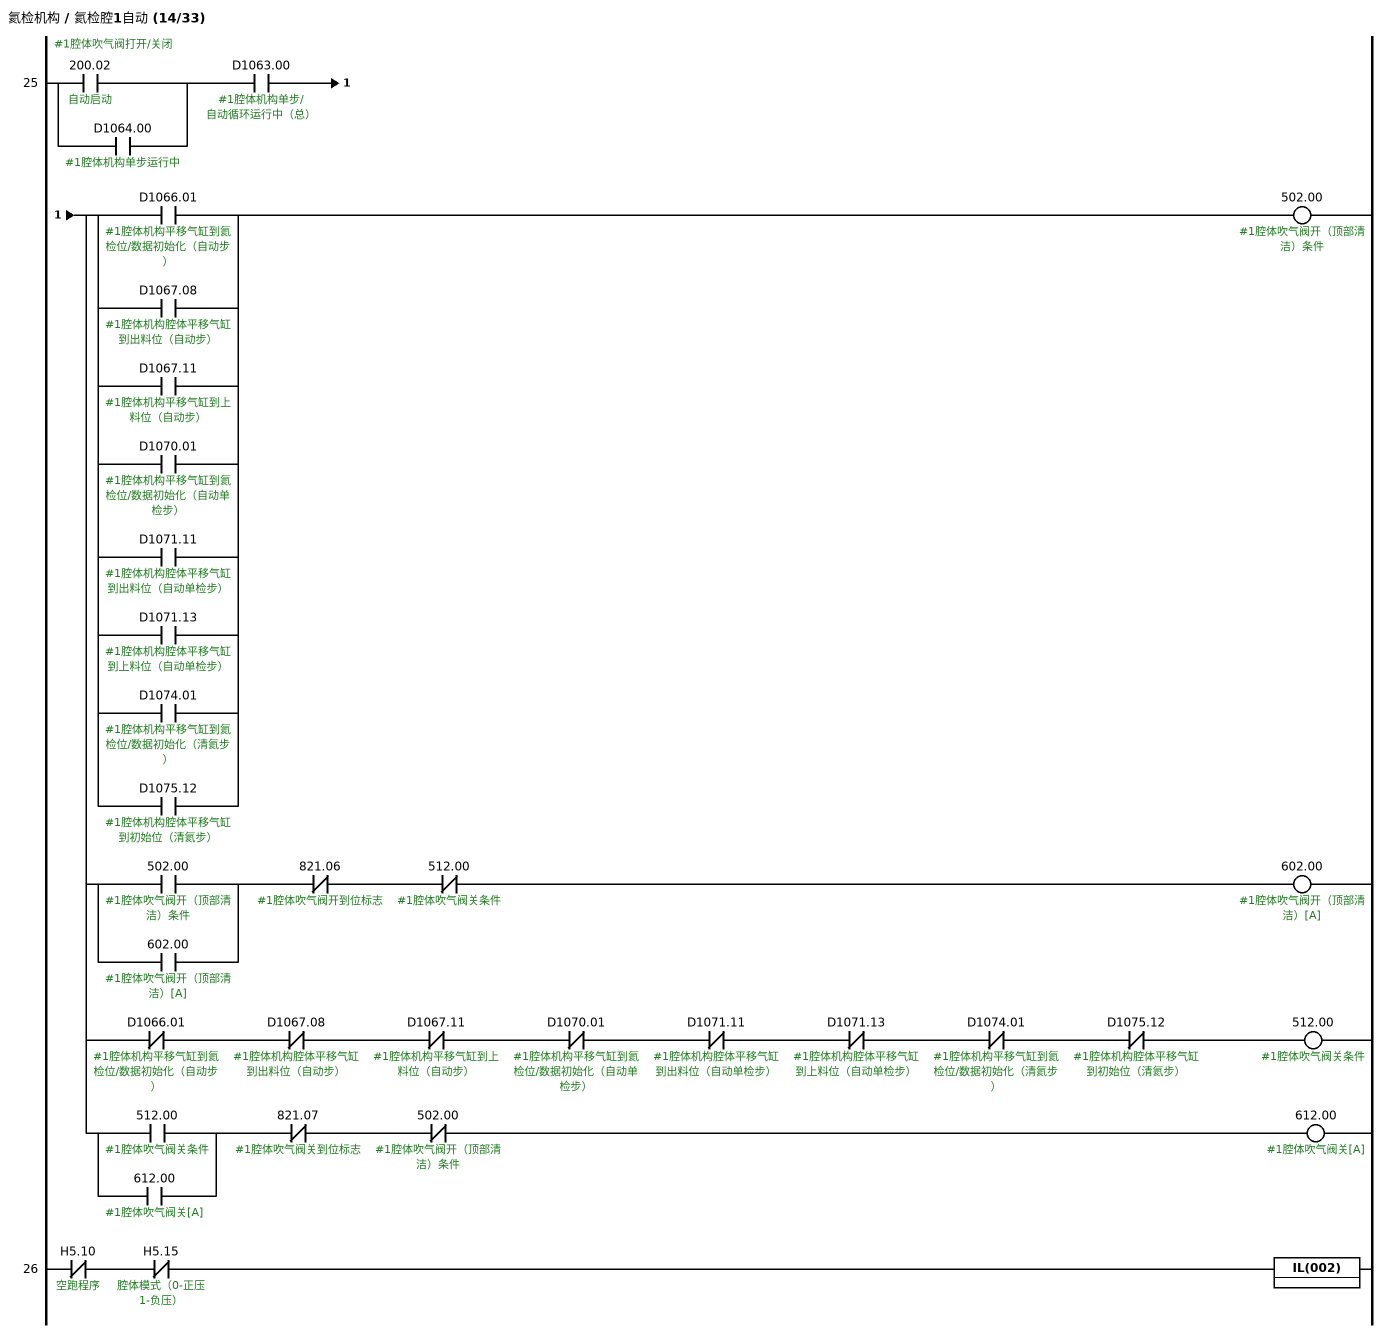
; rung 25: #1腔体吹气阀打开/关闭
LD 200.02  ; 自动启动
OR D1064.00  ; #1腔体机构单步运行中
AND D1063.00  ; #1腔体机构单步/自动循环运行中（总）
OUT TR0
LD D1066.01  ; #1腔体机构平移气缸到氦检位/数据初始化（自动步）
OR D1067.08  ; #1腔体机构腔体平移气缸到出料位（自动步）
OR D1067.11  ; #1腔体机构平移气缸到上料位（自动步）
OR D1070.01  ; #1腔体机构平移气缸到氦检位/数据初始化（自动单检步）
OR D1071.11  ; #1腔体机构腔体平移气缸到出料位（自动单检步）
OR D1071.13  ; #1腔体机构腔体平移气缸到上料位（自动单检步）
OR D1074.01  ; #1腔体机构平移气缸到氦检位/数据初始化（清氦步）
OR D1075.12  ; #1腔体机构腔体平移气缸到初始位（清氦步）
ANDLD
OUT 502.00  ; #1腔体吹气阀开（顶部清洁）条件
LD TR0
LD 502.00  ; #1腔体吹气阀开（顶部清洁）条件
OR 602.00  ; #1腔体吹气阀开（顶部清洁）[A]
ANDLD
ANDNOT 821.06  ; #1腔体吹气阀开到位标志
ANDNOT 512.00  ; #1腔体吹气阀关条件
OUT 602.00  ; #1腔体吹气阀开（顶部清洁）[A]
LD TR0
ANDNOT D1066.01  ; #1腔体机构平移气缸到氦检位/数据初始化（自动步）
ANDNOT D1067.08  ; #1腔体机构腔体平移气缸到出料位（自动步）
ANDNOT D1067.11  ; #1腔体机构平移气缸到上料位（自动步）
ANDNOT D1070.01  ; #1腔体机构平移气缸到氦检位/数据初始化（自动单检步）
ANDNOT D1071.11  ; #1腔体机构腔体平移气缸到出料位（自动单检步）
ANDNOT D1071.13  ; #1腔体机构腔体平移气缸到上料位（自动单检步）
ANDNOT D1074.01  ; #1腔体机构平移气缸到氦检位/数据初始化（清氦步）
ANDNOT D1075.12  ; #1腔体机构腔体平移气缸到初始位（清氦步）
OUT 512.00  ; #1腔体吹气阀关条件
LD TR0
LD 512.00  ; #1腔体吹气阀关条件
OR 612.00  ; #1腔体吹气阀关[A]
ANDLD
ANDNOT 821.07  ; #1腔体吹气阀关到位标志
ANDNOT 502.00  ; #1腔体吹气阀开（顶部清洁）条件
OUT 612.00  ; #1腔体吹气阀关[A]
; rung 26
LDNOT H5.10  ; 空跑程序
ANDNOT H5.15  ; 腔体模式（0-正压 1-负压）
IL(002)

